(* CODESYS project GW42_TVD2300068.project

Project tree, tasks and I/O mapping:
  Device : eSMART (Linux), Exor International, version 3.5.12.0
    application Application
      libraries: Standard, * (System); SysCom, * (System)
      task MainTask (cyclic, interval 20 ms, priority 1) calls PLC_PRG
      program PLC_PRG [ST]: ioList1, digitalProcessing, analogProcessing, commReset, alarmOut, alarmInh, smart_ship
      Symbols
      function block fb_alarmEvent [ST]
      global variables GVL1
      function block fb_tankMonitor [ST]
      function block fb_scaling20R [ST]
      function block fb_linScaleR [ST]
      function block sh_2 [ST]
      function block fb_fluctDet [ST]
      function block fb_nonLinScale20 [ST]
      function block fb_h2s [ST]
      function block fb_buzzer [ST]
      function block fb_comAlarm [ST]
      function block fb_tankMonitor_magLt [ST]
      function block commCheck [ST]
    Modbus_COM : Modbus COM, 3S - Smart Software Solutions GmbH, version 3.5.15.0
      Modbus_Master_COM_Port : Modbus Master, COM Port, 3S - Smart Software Solutions GmbH, version 3.5.15.0
          settings: Transmission = 'RTU'; ResponseTimeout = 1000; TimeBetweenFrames = 5; Auto-restart communication = TRUE
        Modbus_Slave_im1 : Modbus Slave, COM Port, 3S - Smart Software Solutions GmbH, version 3.5.15.0
            settings: SlaveAddress = 11; Channel 0.Function Code = 3; Channel 0.Read Offset = 16#0007; Channel 0.Read Length = 1; Channel 0.Write Offset = 0; Channel 0.Write Length = 0; Channel 0.Cycle Time = 100; Channel 1.Function Code = 3; Channel 1.Read Offset = 16#0064; Channel 1.Read Length = 1; Channel 1.Write Offset = 0; Channel 1.Write Length = 0; Channel 1.Cycle Time = 100
            input  im1model : WORD  // Channel 0.Channel 0
            input  w_im1IOstatus : WORD  // Channel 1.Channel 1
            unmapped channels: Channel 0, Channel 1
        Modbus_Slave_im2 : Modbus Slave, COM Port, 3S - Smart Software Solutions GmbH, version 3.5.15.0
            settings: SlaveAddress = 12; Channel 0.Function Code = 3; Channel 0.Read Offset = 16#0007; Channel 0.Read Length = 1; Channel 0.Write Offset = 0; Channel 0.Write Length = 0; Channel 0.Cycle Time = 100; Channel 1.Function Code = 3; Channel 1.Read Offset = 16#0064; Channel 1.Read Length = 1; Channel 1.Write Offset = 0; Channel 1.Write Length = 0; Channel 1.Cycle Time = 100
            input  im2model : WORD  // Channel 0.Channel 0
            input  w_im2IOstatus : WORD  // Channel 1.Channel 1
            unmapped channels: Channel 0, Channel 1
        Modbus_Slave_im3 : Modbus Slave, COM Port, 3S - Smart Software Solutions GmbH, version 3.5.15.0
            settings: SlaveAddress = 13; Channel 0.Function Code = 3; Channel 0.Read Offset = 16#0007; Channel 0.Read Length = 1; Channel 0.Write Offset = 0; Channel 0.Write Length = 0; Channel 0.Cycle Time = 100; Channel 1.Function Code = 3; Channel 1.Read Offset = 16#0064; Channel 1.Read Length = 1; Channel 1.Write Offset = 0; Channel 1.Write Length = 0; Channel 1.Cycle Time = 100
            input  im3model : WORD  // Channel 0.Channel 0
            input  w_im3IOstatus : WORD  // Channel 1.Channel 1
            unmapped channels: Channel 0, Channel 1
        Modbus_Slave_im4 : Modbus Slave, COM Port, 3S - Smart Software Solutions GmbH, version 3.5.15.0
            settings: SlaveAddress = 14; Channel 0.Function Code = 3; Channel 0.Read Offset = 16#0007; Channel 0.Read Length = 1; Channel 0.Write Offset = 0; Channel 0.Write Length = 0; Channel 0.Cycle Time = 100; Channel 1.Function Code = 3; Channel 1.Read Offset = 16#0064; Channel 1.Read Length = 1; Channel 1.Write Offset = 0; Channel 1.Write Length = 0; Channel 1.Cycle Time = 100
            input  im4model : WORD  // Channel 0.Channel 0
            input  w_im4IOstatus : WORD  // Channel 1.Channel 1
            unmapped channels: Channel 0, Channel 1
        Modbus_Slave_im5 : Modbus Slave, COM Port, 3S - Smart Software Solutions GmbH, version 3.5.15.0
            settings: SlaveAddress = 15; Channel 0.Function Code = 3; Channel 0.Read Offset = 16#0007; Channel 0.Read Length = 1; Channel 0.Write Offset = 0; Channel 0.Write Length = 0; Channel 0.Cycle Time = 100; Channel 1.Function Code = 3; Channel 1.Read Offset = 16#0064; Channel 1.Read Length = 1; Channel 1.Write Offset = 0; Channel 1.Write Length = 0; Channel 1.Cycle Time = 100
            input  im5model : WORD  // Channel 0.Channel 0
            input  w_im5IOstatus : WORD  // Channel 1.Channel 1
            unmapped channels: Channel 0, Channel 1
        Modbus_Slave_im6 : Modbus Slave, COM Port, 3S - Smart Software Solutions GmbH, version 3.5.15.0
            settings: SlaveAddress = 16; Channel 0.Function Code = 3; Channel 0.Read Offset = 16#0007; Channel 0.Read Length = 1; Channel 0.Write Offset = 0; Channel 0.Write Length = 0; Channel 0.Cycle Time = 100; Channel 1.Function Code = 3; Channel 1.Read Offset = 16#0064; Channel 1.Read Length = 1; Channel 1.Write Offset = 0; Channel 1.Write Length = 0; Channel 1.Cycle Time = 100
            input  im6model : WORD  // Channel 0.Channel 0
            input  w_im6IOstatus : WORD  // Channel 1.Channel 1
            unmapped channels: Channel 0, Channel 1
        Modbus_Slave_im7 : Modbus Slave, COM Port, 3S - Smart Software Solutions GmbH, version 3.5.15.0
            settings: SlaveAddress = 17; Channel 0.Function Code = 3; Channel 0.Read Offset = 16#0007; Channel 0.Read Length = 1; Channel 0.Write Offset = 0; Channel 0.Write Length = 0; Channel 0.Cycle Time = 100; Channel 1.Function Code = 3; Channel 1.Read Offset = 16#0064; Channel 1.Read Length = 1; Channel 1.Write Offset = 0; Channel 1.Write Length = 0; Channel 1.Cycle Time = 100
            input  im7model : WORD  // Channel 0.Channel 0
            input  w_im7IOstatus : WORD  // Channel 1.Channel 1
            unmapped channels: Channel 0, Channel 1
        Modbus_Slave_om1 : Modbus Slave, COM Port, 3S - Smart Software Solutions GmbH, version 3.5.15.0
            settings: SlaveAddress = 21; ResponseTimeout = 1000; UseExtendedFunctionCodes = TRUE; Channel 0.Function Code = 3; Channel 0.Read Offset = 16#0007; Channel 0.Read Length = 1; Channel 0.Write Offset = 0; Channel 0.Write Length = 0; Channel 0.Cycle Time = 100; Channel 1.Function Code = 6; Channel 1.Read Offset = 0; Channel 1.Read Length = 0; Channel 1.Write Offset = 16#0064; Channel 1.Write Length = 1; Channel 1.Cycle Time = 100
            input  om1model : WORD  // Channel 0.Channel 0
            output w_om1IOStatus : WORD  // Channel 1.Channel 1
            unmapped channels: Channel 0, Channel 1
        Modbus_Slave_aim1 : Modbus Slave, COM Port, 3S - Smart Software Solutions GmbH, version 3.5.15.0
            settings: SlaveAddress = 22; ResponseTimeout = 1000; UseExtendedFunctionCodes = TRUE; Channel 0.Function Code = 3; Channel 0.Read Offset = 16#0007; Channel 0.Read Length = 1; Channel 0.Write Offset = 0; Channel 0.Write Length = 0; Channel 0.Cycle Time = 100; Channel 1.Function Code = 3; Channel 1.Read Offset = 16#0064; Channel 1.Read Length = 16; Channel 1.Write Offset = 0; Channel 1.Write Length = 0; Channel 1.Cycle Time = 100
            input  aim1model : WORD  // Channel 0.Channel 0
            input  w_aim1ch1 : WORD  // Channel 1.Channel 1
            input  w_aim1ch2 : WORD  // Channel 1.Channel 1
            input  w_aim1ch3 : WORD  // Channel 1.Channel 1
            input  w_aim1ch4 : WORD  // Channel 1.Channel 1
            input  w_aim1ch5 : WORD  // Channel 1.Channel 1
            input  w_aim1ch6 : WORD  // Channel 1.Channel 1
            input  w_aim1ch7 : WORD  // Channel 1.Channel 1
            input  w_aim1ch8 : WORD  // Channel 1.Channel 1
            input  w_aim1ch9 : WORD  // Channel 1.Channel 1
            input  w_aim1ch10 : WORD  // Channel 1.Channel 1
            input  w_aim1ch11 : WORD  // Channel 1.Channel 1
            input  w_aim1ch12 : WORD  // Channel 1.Channel 1
            input  w_aim1ch13 : WORD  // Channel 1.Channel 1
            input  w_aim1ch14 : WORD  // Channel 1.Channel 1
            input  w_aim1ch15 : WORD  // Channel 1.Channel 1
            input  w_aim1ch16 : WORD  // Channel 1.Channel 1
            unmapped channels: Channel 0, Channel 1
        Modbus_Slave_iom1 : Modbus Slave, COM Port, 3S - Smart Software Solutions GmbH, version 3.5.15.0
            settings: SlaveAddress = 20; ResponseTimeout = 1000; UseExtendedFunctionCodes = TRUE; Channel 0.Function Code = 3; Channel 0.Read Offset = 16#0007; Channel 0.Read Length = 1; Channel 0.Write Offset = 0; Channel 0.Write Length = 0; Channel 0.Cycle Time = 100; Channel 1.Function Code = 3; Channel 1.Read Offset = 16#0064; Channel 1.Read Length = 1; Channel 1.Write Offset = 0; Channel 1.Write Length = 0; Channel 1.Cycle Time = 100; Channel 2.Function Code = 6; Channel 2.Read Offset = 0; Channel 2.Read Length = 0; Channel 2.Write Offset = 16#0065; Channel 2.Write Length = 1; Channel 2.Cycle Time = 100
            input  iom1model : WORD  // Channel 0.Channel 0
            input  w_iom1Istatus : WORD  // Channel 1.Channel 1
            output w_iom1OStatus : WORD  // Channel 2.Channel 2
            unmapped channels: Channel 0, Channel 1, Channel 2
        Modbus_Slave_im9 : Modbus Slave, COM Port, 3S - Smart Software Solutions GmbH, version 3.5.15.0
            settings: SlaveAddress = 19; ResponseTimeout = 1000; UseExtendedFunctionCodes = TRUE; Channel 0.Function Code = 3; Channel 0.Read Offset = 16#0007; Channel 0.Read Length = 1; Channel 0.Write Offset = 0; Channel 0.Write Length = 0; Channel 0.Cycle Time = 100; Channel 1.Function Code = 3; Channel 1.Read Offset = 16#0064; Channel 1.Read Length = 1; Channel 1.Write Offset = 0; Channel 1.Write Length = 0; Channel 1.Cycle Time = 100
            input  im9model : WORD  // Channel 0.Channel 0
            input  w_im9IOstatus : WORD  // Channel 1.Channel 1
            unmapped channels: Channel 0, Channel 1
        Modbus_Slave_im8 : Modbus Slave, COM Port, 3S - Smart Software Solutions GmbH, version 3.5.15.0
            settings: SlaveAddress = 18; ResponseTimeout = 1000; UseExtendedFunctionCodes = TRUE; Channel 0.Function Code = 3; Channel 0.Read Offset = 16#0007; Channel 0.Read Length = 1; Channel 0.Write Offset = 0; Channel 0.Write Length = 0; Channel 0.Cycle Time = 100; Channel 1.Function Code = 3; Channel 1.Read Offset = 16#0064; Channel 1.Read Length = 1; Channel 1.Write Offset = 0; Channel 1.Write Length = 0; Channel 1.Cycle Time = 100
            input  im8model : WORD  // Channel 0.Channel 0
            input  w_im8IOstatus : WORD  // Channel 1.Channel 1
            unmapped channels: Channel 0, Channel 1
    Ethernet : Ethernet, 3S - Smart Software Solutions GmbH, version 3.5.15.0
        settings: IPAddress = [192,168,2,141]; SubnetMask = [255,255,255,0]; GatewayAddress = [0,0,0,0]; MACAddress = [16#00,16#30,16#D8,16#0D,16#B1,16#39]; NetworkInterfaceName = 'eth0'; NetworkInterfaceName = "eth0"; SaveCommunicationSettings = FALSE
      ModbusTCP_Slave_Device : ModbusTCP Slave Device, 3S - Smart Software Solutions GmbH, version 3.5.15.0
          settings: Unit-ID = 1
          output JB1_DATA : WORD  // Outputs.Outputs
          output JB2_DATA : WORD  // Outputs.Outputs
          output JB3_DATA : WORD  // Outputs.Outputs
          output JB4_DATA : WORD  // Outputs.Outputs
          output JB5_DATA : WORD  // Outputs.Outputs
          output JB6_DATA : WORD  // Outputs.Outputs
          output WH_DATA : WORD  // Outputs.Outputs
          output MP1_DATA : WORD  // Outputs.Outputs
          output MP2_DATA : WORD  // Outputs.Outputs
          output MP3_DATA : WORD  // Outputs.Outputs
          output AI1_DATA : WORD  // Outputs.Outputs
          output AI2_DATA : WORD  // Outputs.Outputs
          output AI3_DATA : WORD  // Outputs.Outputs
          output AI4_DATA : WORD  // Outputs.Outputs
          output AI5_DATA : WORD  // Outputs.Outputs
          output AI6_DATA : WORD  // Outputs.Outputs
          output AI7_DATA : WORD  // Outputs.Outputs
          output AI8_DATA : WORD  // Outputs.Outputs
          output AI9_DATA : WORD  // Outputs.Outputs
          output AI10_DATA : WORD  // Outputs.Outputs
          output AI11_DATA : WORD  // Outputs.Outputs
          output AI12_DATA : WORD  // Outputs.Outputs
          output AI13_DATA : WORD  // Outputs.Outputs
          output AI14_DATA : WORD  // Outputs.Outputs
          output COM_DATA : WORD  // Outputs.Outputs
          unmapped channels: Inputs, Outputs
*)

// Device/Application/GVL1
{attribute 'qualified_only'}
VAR_GLOBAL
	hxi_ack	:	BOOL;
	hxi_silence	:	BOOL;
	hxi_ackEr	:	BOOL;
	hxi_silenceEr	:	BOOL;
	hxi_ackWh	:	BOOL;
	hxi_ackWhOut	:	BOOL;
	hxi_silenceWh	:	BOOL;
	hxi_ackMess	:	BOOL;
	hxi_ackMessOut	:	BOOL;
	hxi_silenceMess	:	BOOL;
	hxo_alarmInd	:	BOOL;
	hxo_alarmIndwh	:	BOOL;
	hxo_alarmIndMess	:	BOOL;
	hxi_alarmInh	:	ARRAY[0..310]	OF	BOOL;
	hxo_inhibited	:	BOOL;
	hwo_inhibited	:	WORD;
	hxi_enginesd_accept: BOOL;
	hxi_enginesd_overide: BOOL;
	hwi_override :WORD;
	enginesd_cd: TIME;
    hxi_inhbit_doors: BOOL;
	Hbo_HMITest: BOOL;
	Hbi_HMI1Resp: BOOL;
	Hbi_HMI2Resp: BOOL;
	Hbi_HMI3Resp: BOOL;
	(**)
	pwi_digitalInputs		: ARRAY[0..12]	OF	WORD;
	pwo_digitalOutputs		: ARRAY[0..4] OF WORD;
	hwi_digAlarmSet		: ARRAY[0..12]	OF	WORD;
	hwi_digAlarmDelay0	: ARRAY[0..15] OF WORD;
	hwi_digAlarmDelay1	: ARRAY[0..15] OF WORD;
	hwi_digAlarmDelay2	: ARRAY[0..15] OF WORD;
	hwi_digAlarmDelay3	: ARRAY[0..15] OF WORD;
	hwi_digAlarmDelay4	: ARRAY[0..15] OF WORD;
	hwi_digAlarmDelay5	: ARRAY[0..15] OF WORD;
	hwi_digAlarmDelay6	: ARRAY[0..15] OF WORD;
	hwi_digAlarmDelay7	: ARRAY[0..15] OF WORD;
	hwi_digAlarmDelay8	: ARRAY[0..15] OF WORD;
	hwi_digAlarmDelay9	: ARRAY[0..15] OF WORD;
	hwi_digAlarmDelay10	: ARRAY[0..15] OF WORD;
	hwi_digAlarmDelay11	: ARRAY[0..15] OF WORD;
	hwi_digAlarmDelay12	: ARRAY[0..15] OF WORD;
	hwi_digAlarmInh		: ARRAY[0..12]	OF	WORD;
	hwi_digAlarmOrEvent		: ARRAY[0..12]	OF	WORD;
	hwo_digitalAlarms		: ARRAY[0..12]	OF	WORD;
	hwo_digitalEvents		: ARRAY[0..12]	OF	WORD;
	hwo_digitalAlarmsp		: ARRAY[0..12]	OF	WORD;
	(**)
	pwi_analogInput	: ARRAY[0..15]	OF	WORD;
	hro_ch0OutVal	: ARRAY[0..5] OF REAL;
	hro_ch1OutVal	: ARRAY[0..5] OF REAL;
	hro_ch2OutVal	: ARRAY[0..5] OF REAL;
	hro_ch3OutVal	: ARRAY[0..5] OF REAL;
	hro_ch4OutVal	: ARRAY[0..5] OF REAL;
	hro_ch5OutVal	: ARRAY[0..5] OF REAL;
	hro_ch6OutVal	: ARRAY[0..5] OF REAL;
	hro_ch7OutVal	: ARRAY[0..5] OF REAL;
	hro_ch8OutVal	: ARRAY[0..5] OF REAL;
	hro_ch9OutVal	: ARRAY[0..5] OF REAL;
	hro_ch10OutVal	: ARRAY[0..5] OF REAL;
	hro_ch11OutVal	: ARRAY[0..5] OF REAL;
	hro_ch12OutVal	: ARRAY[0..5] OF REAL;
	hro_ch13OutVal	: ARRAY[0..5] OF REAL;
	hro_ch14OutVal	: ARRAY[0..5] OF REAL;
	hro_ch15OutVal	: ARRAY[0..5] OF REAL;
	(*Analolg channel LIMIT steady alarms AND channel errors TO HMI*)
(*Hwo_AnalogAlm_Ch1G1.0 : Level 1, Hwo_AnalogAlm_Ch1G1.1 : Level 2, Hwo_AnalogAlm_Ch1G1.2 : Level 3,Hwo_AnalogAlm_Ch1G1.3 : Cable break,Hwo_AnalogAlm_Ch1G1.4 : Over range*)

	hwo_analogAlm	: ARRAY[0..15]	OF	WORD;
	(*Analolg channel limit pulse alarms and channel errors to HMI*)
(*Hwo_AnalogAlm_Ch1G1.0 : Level 1, Hwo_AnalogAlm_Ch1G1.1 : Level 2, Hwo_AnalogAlm_Ch1G1.2 : Level 3,Hwo_AnalogAlm_Ch1G1.3 : Cable break,Hwo_AnalogAlm_Ch1G1.4 : Over range*)

	hwo_analogAlmP	: ARRAY[0..15]	OF	WORD;
(*Alarm message*)
	hwo_almMsg	: ARRAY[0..15] OF WORD; (*Tanks*)
	(*Analog alarm inhibition*)
(*0:inhL1, 1:inhL2, 2:inhL3, 3:inhCable break, 4:inhOver range, 5:buz en L1, 6:buz en L2, 7:buz en L3, 8:buz en err1, 9:buz en err2, 10:inhL4, 11:buz en L4, 12: Auto filter enable
							13:Fill input sensor min value and range when tank empty, 14: Fill input sensor max value and range when tank full*)
	hwi_chPara	: ARRAY[0..15]	OF	WORD;
(* Prameters of analog limit and eror alarms to HMI *)
(*0:L1Lt, 1:L2Lt, 2:L3Lt, 3:L1delay, 4:L2delay, 5:L3delay,6:Errdelay,
											7:ErrFactor, 8:SensorValMin,9:SensorValMax, 10:SensorRangeMin, 11:SensorRangeMax, 12:filterVal, 
											13:L4Lt, 14:L4delay, 15:heightMin, 16:heightMax, 17:density, 18:unusable , 19:height offset in mm, 
											Auto filter-->20: rate of change, 21: sampling time, 22:sample hold time, 23:filter time constant*)
	hri_chSP_Ch0	: ARRAY[0..23] OF REAL;
	hri_chSP_Ch1	: ARRAY[0..23] OF REAL;
	hri_chSP_Ch2	: ARRAY[0..23] OF REAL;
	hri_chSP_Ch3	: ARRAY[0..23] OF REAL;
	hri_chSP_Ch4	: ARRAY[0..23] OF REAL;
	hri_chSP_Ch5	: ARRAY[0..23] OF REAL;
	hri_chSP_Ch6	: ARRAY[0..23] OF REAL;
	hri_chSP_Ch7	: ARRAY[0..23] OF REAL;
	hri_chSP_Ch8	: ARRAY[0..23] OF REAL;
	hri_chSP_Ch9	: ARRAY[0..23] OF REAL;
	hri_chSP_Ch10	: ARRAY[0..23] OF REAL;
	hri_chSP_Ch11	: ARRAY[0..23] OF REAL;
	hri_chSP_Ch12	: ARRAY[0..23] OF REAL;
	hri_chSP_Ch13	: ARRAY[0..23] OF REAL;
	hri_chSP_Ch14	: ARRAY[0..23] OF REAL;
	hri_chSP_Ch15	: ARRAY[0..23] OF REAL;
(*Tank level sampling in*)
	hwi_ch0X	: ARRAY[0..20] OF WORD;
	hwi_ch1X	: ARRAY[0..20] OF WORD;
	hwi_ch2X	: ARRAY[0..20] OF WORD;
	hwi_ch3X	: ARRAY[0..20] OF WORD;
	hwi_ch4X	: ARRAY[0..20] OF WORD;	
	hwi_ch5X	: ARRAY[0..20] OF WORD;	
	hwi_ch6X	: ARRAY[0..20] OF WORD;	
	hwi_ch7X	: ARRAY[0..20] OF WORD;	
	hwi_ch8X	: ARRAY[0..20] OF WORD;	
	hwi_ch9X	: ARRAY[0..20] OF WORD;	
	hwi_ch10X	: ARRAY[0..20] OF WORD;	
	hwi_ch11X	: ARRAY[0..20] OF WORD;	
	hwi_ch12X	: ARRAY[0..20] OF WORD;	
	hwi_ch13X	: ARRAY[0..20] OF WORD;	
	hwi_ch14X	: ARRAY[0..20] OF WORD;	
	hwi_ch15X	: ARRAY[0..20] OF WORD;	
(*Tank level sampling out*)
	hwi_ch0Y	: ARRAY[0..20] OF WORD;
	hwi_ch1Y	: ARRAY[0..20] OF WORD;
	hwi_ch2Y	: ARRAY[0..20] OF WORD;
	hwi_ch3Y	: ARRAY[0..20] OF WORD;
	hwi_ch4Y	: ARRAY[0..20] OF WORD;
	hwi_ch5Y	: ARRAY[0..20] OF WORD;
	hwi_ch6Y	: ARRAY[0..20] OF WORD;
	hwi_ch7Y	: ARRAY[0..20] OF WORD;
	hwi_ch8Y	: ARRAY[0..20] OF WORD;
	hwi_ch9Y	: ARRAY[0..20] OF WORD;
	hwi_ch10Y	: ARRAY[0..20] OF WORD;
	hwi_ch11Y	: ARRAY[0..20] OF WORD;	
	hwi_ch12Y	: ARRAY[0..20] OF WORD;	
	hwi_ch13Y	: ARRAY[0..20] OF WORD;	
	hwi_ch14Y	: ARRAY[0..20] OF WORD;	
	hwi_ch15Y	: ARRAY[0..20] OF WORD;			

END_VAR

// Device/Application/PLC_PRG
PROGRAM PLC_PRG
VAR
	w_modelNo1 : WORD;
	w_modelNo2 : WORD;
	w_modelNo3 : WORD;
	(**)
	aeGroup0: fb_alarmEvent;
	aeGroup1: fb_alarmEvent;
	aeGroup2: fb_alarmEvent;
	aeGroup3: fb_alarmEvent;
	aeGroup4: fb_alarmEvent;
	aeGroup5: fb_alarmEvent;
	aeGroup6: fb_alarmEvent;
	aeGroup7: fb_alarmEvent;
	aeGroup8: fb_alarmEvent;
	aeGroup9: fb_alarmEvent;
	aeGroup10: fb_alarmEvent;
	aeGroup11: fb_alarmEvent;
	aeGroup12: fb_alarmEvent;
	
	w_digAlarmInh		: ARRAY[0..12]	OF	WORD;
	w_anaAlarmInh		: ARRAY[0..15]	OF	WORD;
	lwi_interlocks		: ARRAY[0..12]	OF	WORD;
	lx_refresh: BOOL;
	lx_ack: BOOL;
	lwo_dialmBuzzer: WORD;
	lwo_dialmInd: WORD;
	(**)
	tmGroup0: fb_tankMonitor;	
	tmGroup1: fb_tankMonitor;
	tmGroup2: fb_tankMonitor;
	tmGroup3: fb_tankMonitor;
	tmGroup4: fb_tankMonitor;
	tmGroup5: fb_tankMonitor;
	tmGroup6: fb_tankMonitor;
	tmGroup7: fb_tankMonitor;
	tmGroup8: fb_tankMonitor;
	tmGroup9: fb_tankMonitor;
	tmGroup10: fb_tankMonitor;
	tmGroup11: fb_tankMonitor;	
	tmGroup12: fb_tankMonitor;
	tmGroup13: fb_tankMonitor;
	tmGroup14: fb_tankMonitor;
	tmGroup15: fb_tankMonitor;	
	lwo_aialmBuzzer: WORD;
	lwo_aialmInd: WORD;
	
	
(*commReset*)	
	x_im1Error : BOOL;
	im1Errorcode : MB_ErrorCodes;
	x_im1Ack: BOOL;

	x_masterReset: BOOL;
	x_im1Reset: BOOL;
	x_im2Reset: BOOL;
	x_im3Reset: BOOL;
	x_im4Reset: BOOL;
	x_im5Reset: BOOL;
	x_im6Reset: BOOL;
	x_im7Reset: BOOL;
	x_im8Reset: BOOL;
	x_om1Reset: BOOL;
	x_aim1Reset: BOOL;	
	
	ton_blink1: TON;
	ton_blink2: TON;
	ton_blink3: TON;
	ton_blink4: TON;
	ton_blink5: TON;
	ton_blink6: TON;
	ton_blink7: TON;
	ton_blink8: TON;
	ton_blink9: TON;
	ton_blink11: TON;
	ton_blink12: TON;
	ton_blink13: TON;
	ton_blink14: TON;
	ton_blink15: TON;
	ton_blink16: TON;
	ton_blink17: TON;
	ton_blink18: TON;
	ton_blink19: TON;
	ton_blink20: TON;
	ton_blink21: TON;	
	ton_blink22: TON;
	
	tp_blink1: TP;
	tp_blink2: TP;
	tp_blink3: TP;
	tp_blink4: TP;
	tp_blink5: TP;
	tp_blink6: TP;
	tp_blink7: TP;
	tp_blink8: TP;
	tp_blink9: TP;
	tp_blink10: TP;
	tp_blink11: TP;
	tp_blink12: TP;
	tp_blink13: TP;
	tp_blink14: TP;
	tp_blink15: TP;
	tp_blink16: TP;
	tp_blink17: TP;
	tp_blink18: TP;
	tp_blink19: TP;
	tp_blink20: TP;
	tp_blink21: TP;
	tp_blink22: TP;
	

	x_mbReset: BOOL;
(*Alarm out*)
	buzzerSet1: fb_buzzer;
	buzzerSet2: fb_buzzer;
	buzzerSet3: fb_buzzer;
	buzzerSet4: fb_buzzer;
	buzzerSet5: fb_buzzer;
    buzzerSet6: fb_buzzer;			
	comAlarm: fb_comAlarm;
	comAlarm1: fb_comAlarm;
	comAlarm2: fb_comAlarm;	
commCheck1: commCheck;
	ee: fb_tankMonitor;
	ton_enginesd: TON;
	
	
	
	overide_out: BOOL;
	poweron_ton: TON;
	wi_interlocks: INT;
END_VAR

w_modelNo1 := im1model;

ioList1();
digitalProcessing();
analogProcessing();
alarmOut();
commReset();
alarmInh();
smart_ship();

ACTION ioList1:
//Digital input module JB1 - S3306: 16CH							
GVL1.Pwi_DigitalInputs[0].0	 := NOT w_im1IOStatus.0	AND NOT GVL1.hwo_digitalAlarms[12].0	;	(*	DI:01	GEN.ROOM PORT BILGE ALARM	*)
GVL1.Pwi_DigitalInputs[0].1	 := NOT w_im1IOStatus.1	AND NOT GVL1.hwo_digitalAlarms[12].0	;	(*	DI:02	PORT GEN EXHAUST TEMP HIGH	*)
GVL1.Pwi_DigitalInputs[0].2	 := NOT w_im1IOStatus.2	AND NOT GVL1.hwo_digitalAlarms[12].0	;	(*	DI:03	PORT GENERATOR COMMON ALARM	*)
GVL1.Pwi_DigitalInputs[0].3	 := NOT w_im1IOStatus.3	AND NOT GVL1.hwo_digitalAlarms[12].0	;	(*	DI:04	PORT GENERATOR RUNNING INDICATION	*)
GVL1.Pwi_DigitalInputs[0].4	 := NOT w_im1IOStatus.4	AND NOT GVL1.hwo_digitalAlarms[12].0	;	(*	DI:05	A.FOULING ALARM: DG(P) & EMG FIRE.P S/C 	*)
GVL1.Pwi_DigitalInputs[0].5	 := NOT w_im1IOStatus.5	AND NOT GVL1.hwo_digitalAlarms[12].0	;	(*	DI:06	STEERING CP: PHASE FAIL MOTOR 1	*)
GVL1.Pwi_DigitalInputs[0].6	 := NOT w_im1IOStatus.6	AND NOT GVL1.hwo_digitalAlarms[12].0	;	(*	DI:07	STEERING CP: POWER FAIL MOTOR 1	*)
GVL1.Pwi_DigitalInputs[0].7	 := NOT w_im1IOStatus.7	AND NOT GVL1.hwo_digitalAlarms[12].0	;	(*	DI:08	STEERING CP: CONTROL FAIL MOTOR 1	*)
GVL1.Pwi_DigitalInputs[0].8	 := NOT w_im1IOStatus.8	AND NOT GVL1.hwo_digitalAlarms[12].0	;	(*	DI:09	STEERING CP: OVERLOAD MOTOR 1	*)
GVL1.Pwi_DigitalInputs[0].9	 := NOT w_im1IOStatus.9	AND NOT GVL1.hwo_digitalAlarms[12].0	;	(*	DI:10	STEERING CP: PHASE FAIL MOTOR 2	*)
GVL1.Pwi_DigitalInputs[0].10	 := NOT w_im1IOStatus.10	AND NOT GVL1.hwo_digitalAlarms[12].0	;	(*	DI:11	STEERING CP: POWER FAIL MOTOR 2	*)
GVL1.Pwi_DigitalInputs[0].11	 := NOT w_im1IOStatus.11	AND NOT GVL1.hwo_digitalAlarms[12].0	;	(*	DI:12	STEERING CP: CONTROL FAIL MOTOR 2	*)
GVL1.Pwi_DigitalInputs[0].12	 := NOT w_im1IOStatus.12	AND NOT GVL1.hwo_digitalAlarms[12].0	;	(*	DI:13	STEERING CP: OVERLOAD MOTOR 2	*)
GVL1.Pwi_DigitalInputs[0].13	 := NOT w_im1IOStatus.13	AND NOT GVL1.hwo_digitalAlarms[12].0	;	(*	DI:14	STEERING CP: LOW OIL LEVEL ALARM	*)
GVL1.Pwi_DigitalInputs[0].14	 := NOT w_im1IOStatus.14	AND NOT GVL1.hwo_digitalAlarms[12].0	;	(*	DI:15	STEERING CP: HIGH OIL TEMP ALARM	*)
GVL1.Pwi_DigitalInputs[0].15	 := NOT w_im1IOStatus.15	AND NOT GVL1.hwo_digitalAlarms[12].0	;	(*	DI:16	STEERING CP: LOW OIL PRESSURE ALARM	*)
//Digital input module JB2 - S3306: 16CH							
GVL1.Pwi_DigitalInputs[1].0	 := NOT w_im2IOStatus.0	AND NOT GVL1.hwo_digitalAlarms[12].1	;	(*	DI:17	GEN.ROOM STBD BILGE ALARM	*)
GVL1.Pwi_DigitalInputs[1].1	 := NOT w_im2IOStatus.1	AND NOT GVL1.hwo_digitalAlarms[12].1	;	(*	DI:18	ENGINE ROOM AFT WT DOOR	*)
GVL1.Pwi_DigitalInputs[1].2	 := NOT w_im2IOStatus.2	AND NOT GVL1.hwo_digitalAlarms[12].1	;	(*	DI:19	CENTER ME EXHAUST TEMP HIGH	*)
GVL1.Pwi_DigitalInputs[1].3	 := NOT w_im2IOStatus.3	AND NOT GVL1.hwo_digitalAlarms[12].1	;	(*	DI:20	STBD GEN EXHAUST TEMP HIGH	*)
GVL1.Pwi_DigitalInputs[1].4	 := NOT w_im2IOStatus.4	AND NOT GVL1.hwo_digitalAlarms[12].1	;	(*	DI:21	STBD GENERATOR COMMON ALARM	*)
GVL1.Pwi_DigitalInputs[1].5	 := NOT w_im2IOStatus.5	AND NOT GVL1.hwo_digitalAlarms[12].1	;	(*	DI:22	STBD GENERATOR RUNNING INDICATION	*)
GVL1.Pwi_DigitalInputs[1].6	 := NOT w_im2IOStatus.6	AND NOT GVL1.hwo_digitalAlarms[12].1	;	(*	DI:23	STBD ME EXHAUST TEMP HIGH	*)
GVL1.Pwi_DigitalInputs[1].7	 := NOT w_im2IOStatus.7	AND NOT GVL1.hwo_digitalAlarms[12].1	;	(*	DI:24	BOW THRUSTER COMMON ALARM	*)
GVL1.Pwi_DigitalInputs[1].8	 := NOT w_im2IOStatus.8	AND NOT GVL1.hwo_digitalAlarms[12].1	;	(*	DI:25	BOW THRUSTER LOW OIL LEVEL ALARM	*)
GVL1.Pwi_DigitalInputs[1].9	 := NOT w_im2IOStatus.9	AND NOT GVL1.hwo_digitalAlarms[12].1	;	(*	DI:26	BOW THRUSTER HIGH OIL TEMP ALARM	*)
GVL1.Pwi_DigitalInputs[1].10	:= NOT w_im2IOStatus.10	AND NOT GVL1.hwo_digitalAlarms[12].1	;	(*	DI:27	OWS POWER SUPPLY FAILURE	*)
GVL1.Pwi_DigitalInputs[1].11	:= NOT w_im2IOStatus.11	AND NOT GVL1.hwo_digitalAlarms[12].1	;	(*	DI:28	OWS 15 PPM ALARM	*)
GVL1.Pwi_DigitalInputs[1].12	:= NOT w_im2IOStatus.12	AND NOT GVL1.hwo_digitalAlarms[12].1	;	(*	DI:29	DCDB-2 BATTERY BREAKER TRIP ALARM	*)
GVL1.Pwi_DigitalInputs[1].13	:= NOT w_im2IOStatus.13	AND NOT GVL1.hwo_digitalAlarms[12].1	;	(*	DI:30	DCDB-2 EARTH FAULT ALARM	*)
GVL1.Pwi_DigitalInputs[1].14	:= NOT w_im2IOStatus.14	AND NOT GVL1.hwo_digitalAlarms[12].1	;	(*	DI:31	DCDB-2 BATTERY CHARGER FAIL ALARM	*)
GVL1.Pwi_DigitalInputs[1].15	:= NOT w_im2IOStatus.15	AND NOT GVL1.hwo_digitalAlarms[12].1	;	(*	DI:32	DCDB-2 BATTERY DISCHARGE ALARM	*)
//Digital input module JB3 - S3306: 16CH							
GVL1.Pwi_DigitalInputs[2].0	:= NOT w_im3IOStatus.0	AND NOT GVL1.hwo_digitalAlarms[12].2	;	(*	DI:33	PORT STERN TUBE FLOW ALARM	*)
GVL1.Pwi_DigitalInputs[2].1	:= NOT w_im3IOStatus.1	AND NOT GVL1.hwo_digitalAlarms[12].2	;	(*	DI:34	STBD STERN TUBE FLOW ALARM	*)
GVL1.Pwi_DigitalInputs[2].2	:= NOT w_im3IOStatus.2	AND NOT GVL1.hwo_digitalAlarms[12].2	;	(*	DI:35	CENTER STERN TUBE FLOW ALARM	*)
GVL1.Pwi_DigitalInputs[2].3	:= NOT w_im3IOStatus.3	AND NOT GVL1.hwo_digitalAlarms[12].2	;	(*	DI:36	PORT ME EXHAUST TEMP HIGH	*)
GVL1.Pwi_DigitalInputs[2].4	:= NOT w_im3IOStatus.4	AND NOT GVL1.hwo_digitalAlarms[12].2	;	(*	DI:37	A.FOULING ALARM: AUX SW.P & EMG FIRE.P S/C	*)
GVL1.Pwi_DigitalInputs[2].5	:= NOT w_im3IOStatus.5	AND NOT GVL1.hwo_digitalAlarms[12].2	;	(*	DI:38	A.FOULING ALARM: DG(S) S/C	*)
GVL1.Pwi_DigitalInputs[2].6	:= NOT w_im3IOStatus.6	AND NOT GVL1.hwo_digitalAlarms[12].2	;	(*	DI:39	PORT ME/GEN STARTING BATTERY LOW ALARM	*)
GVL1.Pwi_DigitalInputs[2].7	:= NOT w_im3IOStatus.7	AND NOT GVL1.hwo_digitalAlarms[12].2	;	(*	DI:40	STBD ME/GEN STARTING BATTERY LOW ALARM	*)
GVL1.Pwi_DigitalInputs[2].8	:= NOT w_im3IOStatus.8	AND NOT GVL1.hwo_digitalAlarms[12].2	;	(*	DI:41	CENTER ME STARTING BATTERY LOW ALARM	*)
GVL1.Pwi_DigitalInputs[2].9	:= NOT w_im3IOStatus.9	AND NOT GVL1.hwo_digitalAlarms[12].2	;	(*	DI:42	AUX COOLING PUMP-2 RUNNING	*)
GVL1.Pwi_DigitalInputs[2].10	:= NOT w_im3IOStatus.10	AND NOT GVL1.hwo_digitalAlarms[12].2	;	(*	DI:43	AUX COOLING PUMP-2 TRIP	*)
GVL1.Pwi_DigitalInputs[2].11	:= NOT w_im3IOStatus.11	AND NOT GVL1.hwo_digitalAlarms[12].2	;	(*	DI:44	ENG.ROOM AFT BILGE ALARM	*)
GVL1.Pwi_DigitalInputs[2].12	:= NOT w_im3IOStatus.12	AND NOT GVL1.hwo_digitalAlarms[12].2	;	(*	DI:45	ENG.ROOM AFT FLOOD ALARM	*)
GVL1.Pwi_DigitalInputs[2].13	:= NOT w_im3IOStatus.13	AND NOT GVL1.hwo_digitalAlarms[12].2	;	(*	DI:46	SPARE	*)
GVL1.Pwi_DigitalInputs[2].14	:= NOT w_im3IOStatus.14	AND NOT GVL1.hwo_digitalAlarms[12].2	;	(*	DI:47	SPARE	*)
GVL1.Pwi_DigitalInputs[2].15	:= NOT w_im3IOStatus.15	AND NOT GVL1.hwo_digitalAlarms[12].2	;	(*	DI:48	SPARE	*)
//Digital input module JB4 - S3306: 16CH							
GVL1.Pwi_DigitalInputs[3].0	:= NOT w_im4IOStatus.0	AND NOT GVL1.hwo_digitalAlarms[12].3	;	(*	DI:49	ENG.ROOM FWD BILGE ALARM	*)
GVL1.Pwi_DigitalInputs[3].1	:= NOT w_im4IOStatus.1	AND NOT GVL1.hwo_digitalAlarms[12].3	;	(*	DI:50	ENG.ROOM FWD FLOOD ALARM	*)
GVL1.Pwi_DigitalInputs[3].2	:= NOT w_im4IOStatus.2	AND NOT GVL1.hwo_digitalAlarms[12].3	;	(*	DI:51	ENGINE ROOM FWD WT DOOR	*)
GVL1.Pwi_DigitalInputs[3].3	:= NOT w_im4IOStatus.3	AND NOT GVL1.hwo_digitalAlarms[12].3	;	(*	DI:52	PROPULSION SYSTEM POWER SUPPLY FAIL	*)
GVL1.Pwi_DigitalInputs[3].4	:= NOT w_im4IOStatus.4	AND NOT GVL1.hwo_digitalAlarms[12].3	;	(*	DI:53	PORT ME PROP.MODULE COMMON ALARM	*)
GVL1.Pwi_DigitalInputs[3].5	:= NOT w_im4IOStatus.5	AND NOT GVL1.hwo_digitalAlarms[12].3	;	(*	DI:54	STBD ME PROP.MODULE COMMON ALARM	*)
GVL1.Pwi_DigitalInputs[3].6	:= NOT w_im4IOStatus.6	AND NOT GVL1.hwo_digitalAlarms[12].3	;	(*	DI:55	CENTER ME PROP.MODULE COMMON ALARM	*)
GVL1.Pwi_DigitalInputs[3].7	:= NOT w_im4IOStatus.7	AND NOT GVL1.hwo_digitalAlarms[12].3	;	(*	DI:56	A.FOULING ALARM: PORT ME & STBD ME S/C	*)
GVL1.Pwi_DigitalInputs[3].8	:= NOT w_im4IOStatus.8	AND NOT GVL1.hwo_digitalAlarms[12].3	;	(*	DI:57	A.FOULING ALARM: CENETR ME S/C	*)
GVL1.Pwi_DigitalInputs[3].9	:= NOT w_im4IOStatus.9	AND NOT GVL1.hwo_digitalAlarms[12].3	;	(*	DI:58	A.FOULING ALARM: SW DOMESTIC & A/C.P SC	*)
GVL1.Pwi_DigitalInputs[3].10	:= NOT w_im4IOStatus.10	AND NOT GVL1.hwo_digitalAlarms[12].3	;	(*	DI:59	ENG.ROOM CO2 RELEASE EAVC ALARM	*)
GVL1.Pwi_DigitalInputs[3].11	:= NOT w_im4IOStatus.11	AND NOT GVL1.hwo_digitalAlarms[12].3	;	(*	DI:60	GEN.ROOM CO2 RELEASE EVAC ALARM	*)
GVL1.Pwi_DigitalInputs[3].12	:= NOT w_im4IOStatus.12	AND NOT GVL1.hwo_digitalAlarms[12].3	;	(*	DI:61	CO2 LEAKAGE ALARM	*)
GVL1.Pwi_DigitalInputs[3].13	:= NOT w_im4IOStatus.13	AND NOT GVL1.hwo_digitalAlarms[12].3	;	(*	DI:62	ENG ROOM CO2 RELEASED ALARM	*)
GVL1.Pwi_DigitalInputs[3].14	:= NOT w_im4IOStatus.14	AND NOT GVL1.hwo_digitalAlarms[12].3	;	(*	DI:63	GEN ROOM CO2 RELEASED ALARM	*)
GVL1.Pwi_DigitalInputs[3].15	:= NOT w_im4IOStatus.15	AND NOT GVL1.hwo_digitalAlarms[12].3	;	(*	DI:64	CO2 SYSTEM POWER FAIL ALARM	*)
//Digital input module JB5 - S3306: 16CH							
GVL1.Pwi_DigitalInputs[4].0	:= NOT w_im5IOStatus.0	AND NOT GVL1.hwo_digitalAlarms[12].4	;	(*	DI:65	PUMP ROOM AFT PORT BILGE ALARM	*)
GVL1.Pwi_DigitalInputs[4].1	:= NOT w_im5IOStatus.1	AND NOT GVL1.hwo_digitalAlarms[12].4	;	(*	DI:66	PUMP ROOM AFT STBD BILGE ALARM	*)
GVL1.Pwi_DigitalInputs[4].2	:= NOT w_im5IOStatus.2	AND NOT GVL1.hwo_digitalAlarms[12].4	;	(*	DI:67	V.SPACE PUMP ROOM FWD (P) BILGE ALARM	*)
GVL1.Pwi_DigitalInputs[4].3	:= NOT w_im5IOStatus.3	AND NOT GVL1.hwo_digitalAlarms[12].4	;	(*	DI:68	V.SPACE PUMP ROOM FWD (S) BILGE ALARM	*)
GVL1.Pwi_DigitalInputs[4].4	:= NOT w_im5IOStatus.4	AND NOT GVL1.hwo_digitalAlarms[12].4	;	(*	DI:69	ACCOM.AREA AFT BILGE ALARM	*)
GVL1.Pwi_DigitalInputs[4].5	:= NOT w_im5IOStatus.5	AND NOT GVL1.hwo_digitalAlarms[12].4	;	(*	DI:70	PUMP ROOM FWD WT DOOR	*)
GVL1.Pwi_DigitalInputs[4].6	:= NOT w_im5IOStatus.6	AND NOT GVL1.hwo_digitalAlarms[12].4	;	(*	DI:71	STP OVERFLOW ALARM	*)
GVL1.Pwi_DigitalInputs[4].7	:= NOT w_im5IOStatus.7	AND NOT GVL1.hwo_digitalAlarms[12].4	;	(*	DI:72	A/C SYSTEM COMMON ALARM	*)
GVL1.Pwi_DigitalInputs[4].8	:= NOT w_im5IOStatus.8	AND NOT GVL1.hwo_digitalAlarms[12].4	;	(*	DI:73	ACCOM.AREA FWD BILGE ALARM	*)
GVL1.Pwi_DigitalInputs[4].9	:= NOT w_im5IOStatus.9	AND NOT GVL1.hwo_digitalAlarms[12].4	;	(*	DI:74	FWD PASSAGE BILGE ALARM	*)
GVL1.Pwi_DigitalInputs[4].10	:= NOT w_im5IOStatus.10	AND NOT GVL1.hwo_digitalAlarms[12].4	;	(*	DI:75	FOREPEAK COMPT BILGE ALARM	*)
GVL1.Pwi_DigitalInputs[4].11	:= NOT w_im5IOStatus.11	AND NOT GVL1.hwo_digitalAlarms[12].4	;	(*	DI:76	ACCOM.AREA WT DOOR	*)
GVL1.Pwi_DigitalInputs[4].12	:= NOT w_im5IOStatus.12	AND NOT GVL1.hwo_digitalAlarms[12].4	;	(*	DI:77	A/C FIRE DAMPER CLOSED ALARM	*)
GVL1.Pwi_DigitalInputs[4].13	:= NOT w_im5IOStatus.13	AND NOT GVL1.hwo_digitalAlarms[12].4	;	(*	DI:78	GALLEY VENT OUT FIRE DAMPER CLOSED ALARM	*)
GVL1.Pwi_DigitalInputs[4].14	:= NOT w_im5IOStatus.14	AND NOT GVL1.hwo_digitalAlarms[12].4	;	(*	DI:79	GALLEY VENT IN FIRE DAMPER CLOSED ALARM	*)
GVL1.Pwi_DigitalInputs[4].15	:= NOT w_im5IOStatus.15	AND NOT GVL1.hwo_digitalAlarms[12].4	;	(*	DI:80	GALLEY HD VENT FIRE DAMPER CLOSED ALARM	*)

//Digital input module JB6 - S3306: 16CH							
GVL1.Pwi_DigitalInputs[5].0	:= NOT w_im6IOStatus.0	AND NOT GVL1.hwo_digitalAlarms[12].5	;	(*	DI:81	DCDB1 SEC-1 BAT.CHARGER FAILURE ALARM	*)
GVL1.Pwi_DigitalInputs[5].1	:= NOT w_im6IOStatus.1	AND NOT GVL1.hwo_digitalAlarms[12].5	;	(*	DI:82	DCDB1 SEC-1 BAT. DISCHARGE ALARM	*)
GVL1.Pwi_DigitalInputs[5].2	:= NOT w_im6IOStatus.2	AND NOT GVL1.hwo_digitalAlarms[12].5	;	(*	DI:83	DCDB1 SEC-1 BAT. LOW VOLT ALARM	*)
GVL1.Pwi_DigitalInputs[5].3	:= NOT w_im6IOStatus.3	AND NOT GVL1.hwo_digitalAlarms[12].5	;	(*	DI:84	DCDB1 SEC-1 BAT. BANK CB TRIP ALARM	*)
GVL1.Pwi_DigitalInputs[5].4	:= NOT w_im6IOStatus.4	AND NOT GVL1.hwo_digitalAlarms[12].5	;	(*	DI:85	DCDB1 SEC-2 BAT.CHARGER FAILURE ALARM	*)
GVL1.Pwi_DigitalInputs[5].5	:= NOT w_im6IOStatus.5	AND NOT GVL1.hwo_digitalAlarms[12].5	;	(*	DI:86	DCDB1 SEC-2 BAT. DISCHARGE ALARM	*)
GVL1.Pwi_DigitalInputs[5].6	:= NOT w_im6IOStatus.6	AND NOT GVL1.hwo_digitalAlarms[12].5	;	(*	DI:87	DCDB1 SEC-2 BAT. LOW VOLT ALARM	*)
GVL1.Pwi_DigitalInputs[5].7	:= NOT w_im6IOStatus.7	AND NOT GVL1.hwo_digitalAlarms[12].5	;	(*	DI:88	DCDB1 SEC-2 BAT. BANK CB TRIP ALARM	*)
GVL1.Pwi_DigitalInputs[5].8	:= NOT w_im6IOStatus.8	AND NOT GVL1.hwo_digitalAlarms[12].5	;	(*	DI:89	SEC-1 AND SEC-2 EARTH FAULT	*)
GVL1.Pwi_DigitalInputs[5].9	:= NOT w_im6IOStatus.9	AND NOT GVL1.hwo_digitalAlarms[12].5	;	(*	DI:90	FREEZER CTRL PANEL COMMON ALARM	*)
GVL1.Pwi_DigitalInputs[5].10	:= NOT w_im6IOStatus.10	AND NOT GVL1.hwo_digitalAlarms[12].5	;	(*	DI:91	CHILLER CTRL PANEL COMMON ALARM	*)
GVL1.Pwi_DigitalInputs[5].11	:= NOT w_im6IOStatus.11	AND NOT GVL1.hwo_digitalAlarms[12].5	;	(*	DI:92	MAN TRAP ALARM: FREEZER ROOM	*)
GVL1.Pwi_DigitalInputs[5].12	:= NOT w_im6IOStatus.12	AND NOT GVL1.hwo_digitalAlarms[12].5	;	(*	DI:93	MAN TRAP ALARM: CHILLER ROOM	*)
GVL1.Pwi_DigitalInputs[5].13	:= NOT w_im6IOStatus.13	AND NOT GVL1.hwo_digitalAlarms[12].5	;	(*	DI:94	PUMP RM COMP. AREA AREA REF. LEAKAGE ALARM 	*)
GVL1.Pwi_DigitalInputs[5].14	:= NOT w_im6IOStatus.14	AND NOT GVL1.hwo_digitalAlarms[12].5	;	(*	DI:95	BELOW DECK. AREA AREA REF. LEAKAGE ALARM 	*)
GVL1.Pwi_DigitalInputs[5].15	:= NOT w_im6IOStatus.15	AND NOT GVL1.hwo_digitalAlarms[12].5	;	(*	DI:96	CO2 ROOM FAN TRIP ALARM	*)
//Digital input module WH - S3306: 16CH							
GVL1.Pwi_DigitalInputs[6].0	:= NOT w_im7IOStatus.0	AND NOT GVL1.hwo_digitalAlarms[12].6	;	(*	DI:97	WH ALARM MUTE P/B	*)
GVL1.Pwi_DigitalInputs[6].1	:= NOT w_im7IOStatus.1	AND NOT GVL1.hwo_digitalAlarms[12].6	;	(*	DI:98	STGR JOYSTICK CONTROL FAIL ALARM	*)
GVL1.Pwi_DigitalInputs[6].2	:= NOT w_im7IOStatus.2	AND NOT GVL1.hwo_digitalAlarms[12].6	;	(*	DI:99	GEN.ALARM MAIN SUPPLY FAILURE	*)
GVL1.Pwi_DigitalInputs[6].3	:= NOT w_im7IOStatus.3	AND NOT GVL1.hwo_digitalAlarms[12].6	;	(*	DI:100	GEN.ALARM ALT.SUPPLY FAILURE	*)
GVL1.Pwi_DigitalInputs[6].4	:= NOT w_im7IOStatus.4	AND NOT GVL1.hwo_digitalAlarms[12].6	;	(*	DI:101	NAV.LIGHT POWER FAILURE	*)
GVL1.Pwi_DigitalInputs[6].5	:= NOT w_im7IOStatus.5	AND NOT GVL1.hwo_digitalAlarms[12].6	;	(*	DI:102	NAV.LIGHT SYSTEM FAULT	*)
GVL1.Pwi_DigitalInputs[6].6	:= NOT w_im7IOStatus.6	AND NOT GVL1.hwo_digitalAlarms[12].6	;	(*	DI:103	FIRE ALARM SYSTEM FAULT	*)
GVL1.Pwi_DigitalInputs[6].7	:= NOT w_im7IOStatus.7	AND NOT GVL1.hwo_digitalAlarms[12].6	;	(*	DI:104	FIRE ALARM ACTVATED	*)
GVL1.Pwi_DigitalInputs[6].8	:= NOT w_im7IOStatus.8	AND NOT GVL1.hwo_digitalAlarms[12].6	;	(*	DI:105	AUTO PILOT FAIL ALARM	*)
GVL1.Pwi_DigitalInputs[6].9	:= NOT w_im7IOStatus.9	AND NOT GVL1.hwo_digitalAlarms[12].6	;	(*	DI:106	GAS DETECTION SYSTEM POWER FAIL	*)
GVL1.Pwi_DigitalInputs[6].10	:= NOT w_im7IOStatus.10	AND NOT GVL1.hwo_digitalAlarms[12].6	;	(*	DI:107	H2S ALARM ACTIVATED	*)
GVL1.Pwi_DigitalInputs[6].11	:= NOT w_im7IOStatus.11	AND NOT GVL1.hwo_digitalAlarms[12].6	;	(*	DI:108	LEL ALARM ACTIVATED	*)
GVL1.Pwi_DigitalInputs[6].12	:= NOT w_im7IOStatus.12	AND NOT GVL1.hwo_digitalAlarms[12].6	;	(*	DI:109	WH AREA REF. LEAKAGE ALARM 	*)
GVL1.Pwi_DigitalInputs[6].13	:= NOT w_im7IOStatus.13	AND NOT GVL1.hwo_digitalAlarms[12].6	;	(*	DI:110	PASSENGER AREA REF. LEAKAGE ALARM 	*)
GVL1.Pwi_DigitalInputs[6].14	:= NOT w_im7IOStatus.14	AND NOT GVL1.hwo_digitalAlarms[12].6	;	(*	DI:111	DEPTH BELOW KEEL LOWER THAN SET.P 	*)
GVL1.Pwi_DigitalInputs[6].15	:= NOT w_im7IOStatus.15	AND NOT GVL1.hwo_digitalAlarms[12].6	;	(*	DI:112	GMDSS COMMON ALRM	*)
//Digital input module1  MP- S3306: 16CH							
GVL1.Pwi_DigitalInputs[7].0	:= NOT w_im8IOstatus.0	AND NOT GVL1.hwo_digitalAlarms[12].7	;	(*	DI:113	PORT ME COMMON ALARM	*)
GVL1.Pwi_DigitalInputs[7].1	:= NOT w_im8IOstatus.1	AND NOT GVL1.hwo_digitalAlarms[12].7	;	(*	DI:114	STBD ME COMMON ALARM	*)
GVL1.Pwi_DigitalInputs[7].2	:= NOT w_im8IOstatus.2	AND NOT GVL1.hwo_digitalAlarms[12].7	;	(*	DI:115	CENTER ME COMMON ALARM	*)
GVL1.Pwi_DigitalInputs[7].3	:= NOT w_im8IOstatus.3	AND NOT GVL1.hwo_digitalAlarms[12].7	;	(*	DI:116	AUX COOLING PUMP-1 RUNNING	*)
GVL1.Pwi_DigitalInputs[7].4	:= NOT w_im8IOstatus.4	AND NOT GVL1.hwo_digitalAlarms[12].7	;	(*	DI:117	AUX COOLING PUMP-1 TRIP	*)
GVL1.Pwi_DigitalInputs[7].5	:= NOT w_im8IOstatus.5	AND NOT GVL1.hwo_digitalAlarms[12].7	;	(*	DI:118	FO PURIFIER COMMON ALRM	*)
GVL1.Pwi_DigitalInputs[7].6	:= NOT w_im8IOstatus.6	AND NOT GVL1.hwo_digitalAlarms[12].7	;	(*	DI:119	MSB: PREF. TRIP ALARM	*)
GVL1.Pwi_DigitalInputs[7].7	:= NOT w_im8IOstatus.7	AND NOT GVL1.hwo_digitalAlarms[12].7	;	(*	DI:120	MSB: 440V EARTH FAULT ALARM	*)
GVL1.Pwi_DigitalInputs[7].8	:= NOT w_im8IOstatus.8	AND NOT GVL1.hwo_digitalAlarms[12].7	;	(*	DI:121	MSB: 220V EARTH FAULT ALARM	*)
GVL1.Pwi_DigitalInputs[7].9	:= NOT w_im8IOstatus.9	AND NOT GVL1.hwo_digitalAlarms[12].7	;	(*	DI:122	MSB: 24VDC SUPPLY FAIL ALARM	*)
GVL1.Pwi_DigitalInputs[7].10	:= NOT w_im8IOstatus.10	AND NOT GVL1.hwo_digitalAlarms[12].7	;	(*	DI:123	MSB: ABNORMAL ALARM	*)
GVL1.Pwi_DigitalInputs[7].11	:= NOT w_im8IOstatus.11	AND NOT GVL1.hwo_digitalAlarms[12].7	;	(*	DI:124	AMS AC SUPPLY FAIL	*)
GVL1.Pwi_DigitalInputs[7].12	:= NOT w_im8IOstatus.12	AND NOT GVL1.hwo_digitalAlarms[12].7	;	(*	DI:125	AMS DC SUPPLY FAIL	*)
GVL1.Pwi_DigitalInputs[7].13	:= NOT w_im8IOstatus.13	AND NOT GVL1.hwo_digitalAlarms[12].7	;	(*	DI:126	ALRM MUTE AMS PANEL	*)
GVL1.Pwi_DigitalInputs[7].14	:= NOT w_im8IOstatus.14	AND NOT GVL1.hwo_digitalAlarms[12].7	;	(*	DI:127	SPARE	*)
GVL1.Pwi_DigitalInputs[7].15	:= NOT w_im8IOstatus.15	AND NOT GVL1.hwo_digitalAlarms[12].7	;	(*	DI:128	SPARE	*)
//Digital input module1  MP- S3306: 16CH							
GVL1.Pwi_DigitalInputs[8].0	:= NOT w_im9IOstatus.0	AND NOT GVL1.hwo_digitalAlarms[12].7	;	(*	DI:129	SPARE	*)
GVL1.Pwi_DigitalInputs[8].1	:= NOT w_im9IOstatus.1	AND NOT GVL1.hwo_digitalAlarms[12].7	;	(*	DI:130	SPARE	*)
GVL1.Pwi_DigitalInputs[8].2	:= NOT w_im9IOstatus.2	AND NOT GVL1.hwo_digitalAlarms[12].7	;	(*	DI:131	SPARE	*)
GVL1.Pwi_DigitalInputs[8].3	:= NOT w_im9IOstatus.3	AND NOT GVL1.hwo_digitalAlarms[12].7	;	(*	DI:132	SPARE	*)
GVL1.Pwi_DigitalInputs[8].4	:= NOT w_im9IOstatus.4	AND NOT GVL1.hwo_digitalAlarms[12].7	;	(*	DI:133	SPARE	*)
GVL1.Pwi_DigitalInputs[8].5	:= NOT w_im9IOstatus.5	AND NOT GVL1.hwo_digitalAlarms[12].7	;	(*	DI:134	SPARE	*)
GVL1.Pwi_DigitalInputs[8].6	:= NOT w_im9IOstatus.6	AND NOT GVL1.hwo_digitalAlarms[12].7	;	(*	DI:135	SPARE	*)
GVL1.Pwi_DigitalInputs[8].7	:= NOT w_im9IOstatus.7	AND NOT GVL1.hwo_digitalAlarms[12].7	;	(*	DI:136	SPARE	*)
GVL1.Pwi_DigitalInputs[8].8	:= NOT w_im9IOstatus.8	AND NOT GVL1.hwo_digitalAlarms[12].7	;	(*	DI:137	SPARE	*)
GVL1.Pwi_DigitalInputs[8].9	:= NOT w_im9IOstatus.9	AND NOT GVL1.hwo_digitalAlarms[12].7	;	(*	DI:138	SPARE	*)
GVL1.Pwi_DigitalInputs[8].10	:= NOT w_im9IOstatus.10	AND NOT GVL1.hwo_digitalAlarms[12].7	;	(*	DI:139	SPARE	*)
GVL1.Pwi_DigitalInputs[8].11	:= NOT w_im9IOstatus.11	AND NOT GVL1.hwo_digitalAlarms[12].7	;	(*	DI:140	SPARE	*)
GVL1.Pwi_DigitalInputs[8].12	:= NOT w_im9IOstatus.12	AND NOT GVL1.hwo_digitalAlarms[12].7	;	(*	DI:141	SPARE	*)
GVL1.Pwi_DigitalInputs[8].13	:= NOT w_im9IOstatus.13	AND NOT GVL1.hwo_digitalAlarms[12].7	;	(*	DI:142	SPARE	*)
GVL1.Pwi_DigitalInputs[8].14	:= NOT w_im9IOstatus.14	AND NOT GVL1.hwo_digitalAlarms[12].7	;	(*	DI:143	SPARE	*)
GVL1.Pwi_DigitalInputs[8].15	:= NOT w_im9IOstatus.15	AND NOT GVL1.hwo_digitalAlarms[12].7	;	(*	DI:144	SPARE	*)
//Digital I/O module MP- S3301: 8CH							
GVL1.Pwi_DigitalInputs[9].0	:=  w_iom1IStatus.0	AND NOT GVL1.hwo_digitalAlarms[12].8	;	(*	DI:145	SPARE	*)
GVL1.Pwi_DigitalInputs[9].1	:=  w_iom1IStatus.1	AND NOT GVL1.hwo_digitalAlarms[12].8	;	(*	DI:146	SPARE	*)
GVL1.Pwi_DigitalInputs[9].2	:=  w_iom1IStatus.2	AND NOT GVL1.hwo_digitalAlarms[12].8	;	(*	DI:147	SPARE	*)
GVL1.Pwi_DigitalInputs[9].3	:=  w_iom1IStatus.3	AND NOT GVL1.hwo_digitalAlarms[12].8	;	(*	DI:148	SPARE	*)
GVL1.Pwi_DigitalInputs[9].4	:=  w_iom1IStatus.4	AND NOT GVL1.hwo_digitalAlarms[12].8	;	(*	DI:149	SPARE	*)
GVL1.Pwi_DigitalInputs[9].5	:=  w_iom1IStatus.5	AND NOT GVL1.hwo_digitalAlarms[12].8	;	(*	DI:150	SPARE	*)
GVL1.Pwi_DigitalInputs[9].6	:=  w_iom1IStatus.6	AND NOT GVL1.hwo_digitalAlarms[12].8	;	(*	DI:151	SPARE	*)
GVL1.Pwi_DigitalInputs[9].7	:=  w_iom1IStatus.7	AND NOT GVL1.hwo_digitalAlarms[12].8	;	(*	DI:152	SPARE	*)




						
//Communication alarms - Soft channel: 16Ch					
GVL1.Pwi_DigitalInputs[12].0	 := NOT ton_blink11.Q	;	(*	JB1 DI MODULE COMMS: FAIL	*)
GVL1.Pwi_DigitalInputs[12].1	 := NOT ton_blink12.Q	;	(*	JB2 DI MODULE COMMS: FAIL	*)
GVL1.Pwi_DigitalInputs[12].2	 := NOT ton_blink13.Q	;	(*	JB3 DI MODULE COMMS: FAIL	*)
GVL1.Pwi_DigitalInputs[12].3	 := NOT ton_blink14.Q	;	(*	JB4 DI MODULE COMMS: FAIL	*)
GVL1.Pwi_DigitalInputs[12].4	 := NOT ton_blink15.Q	;	(*	JB5 DI MODULE COMMS: FAIL	*)
GVL1.Pwi_DigitalInputs[12].5	 := NOT ton_blink16.Q	;	(*	JB6 DI MODULE COMMS: FAIL	*)
GVL1.Pwi_DigitalInputs[12].6	 := NOT ton_blink17.Q	;	(*	WH DI MODULE COMMS: FAIL	*)
GVL1.Pwi_DigitalInputs[12].7	 := NOT ton_blink18.Q	;	(*	MP DI1 MODULE COMMS: FAIL	*)
GVL1.Pwi_DigitalInputs[12].8	 := NOT ton_blink19.Q	;	(*	MP DI2 MODULE COMMS: FAIL	*)
GVL1.Pwi_DigitalInputs[12].9	 := NOT ton_blink20.Q	;	(*	MP DIO MODULE COMMS: FAIL	*)
GVL1.Pwi_DigitalInputs[12].10	 := NOT ton_blink21.Q	;	(*	MP DO MODULE COMMS: FAIL	*)
GVL1.Pwi_DigitalInputs[12].11	 := NOT ton_blink22.Q	;	(*	MP AI MODULE COMMS: FAIL	*)
GVL1.Pwi_DigitalInputs[12].12	 := commCheck1.Lbo_ComErr1	; (*	ECR HMI COMMS: FAIL	*)			
GVL1.Pwi_DigitalInputs[12].13	 := commCheck1.Lbo_ComErr2	; (*	WH HMI COMMS: FAIL	*)		
GVL1.Pwi_DigitalInputs[12].14	 := commCheck1.Lbo_ComErr3	; (*	MESS HMI COMMS: FAIL	*)
GVL1.Pwi_DigitalInputs[12].15	 := 0	;			
	
	
			

(*Shore mode interlock for doors*)
lwi_interlocks[1].1 := GVL1.hxi_inhbit_doors;
lwi_interlocks[3].2 := GVL1.hxi_inhbit_doors;
lwi_interlocks[4].5  := GVL1.hxi_inhbit_doors;
lwi_interlocks[4].11  := GVL1.hxi_inhbit_doors;

//Digital IO module1 - S3303E: 8Ch		
w_iom1OStatus.0	 := NOT GVL1.pwo_digitalOutputs[0].0 	;	
w_iom1OStatus.1	 := NOT GVL1.pwo_digitalOutputs[0].1	;	
w_iom1OStatus.2	 := NOT GVL1.pwo_digitalOutputs[0].2	;	
w_iom1OStatus.3	 := NOT GVL1.pwo_digitalOutputs[0].3	;	
w_iom1OStatus.4	 := NOT GVL1.pwo_digitalOutputs[0].4	;	
w_iom1OStatus.5	 := NOT GVL1.pwo_digitalOutputs[0].5	;	



//Digital output module1 - S3303E: 16Ch	
poweron_ton(IN:=TRUE , PT:=T#10S , Q=> , ET=> );	
w_om1IOStatus.0	 := comAlarm.LDo_Accoustic1 AND poweron_ton.Q;	(*	VISUAL & AUDIO ALARM BUZZER ENG: ROOM	*)
w_om1IOStatus.1	 := comAlarm.LDo_Accoustic1 AND poweron_ton.Q;	(*	VISUAL & AUDIO ALARM BUZZER GEN: ROOM	*)
w_om1IOStatus.2	 := comAlarm.LDo_Accoustic1 AND poweron_ton.Q;	(*	VISUAL & AUDIO ALARM BUZZER PUMP ROOM	*)
w_om1IOStatus.3	 := comAlarm2.LDo_Accoustic1 AND poweron_ton.Q;		(*	BUZZER WITH IND MESS ROOM	*)
w_om1IOStatus.4	 := comAlarm1.LDo_Accoustic1 AND poweron_ton.Q;	(*	BUZZER WITH IND WHEEL HOUSE	*)

w_om1IOStatus.5	 := GVL1.pwo_digitalOutputs[1].5	;	(*	GREY WATER TANK LOW AUTO STOP GREY WATER PUMP PUMP	*)
IF GVL1.hwo_analogAlm[3].1 AND NOT GVL1.hwi_override.0 
THEN GVL1.pwo_digitalOutputs[1].5:= 1; ELSE GVL1.pwo_digitalOutputs[1].5:=0;	END_IF

w_om1IOStatus.6	 := GVL1.pwo_digitalOutputs[1].6	;	(*	FUEL TANK HIGH AUTO STOP FO PUMP	*)
IF (GVL1.hwo_analogAlm[4].2 AND NOT GVL1.hwi_override.1) OR (GVL1.hwo_analogAlm[5].2 AND NOT GVL1.hwi_override.2)
OR (GVL1.hwo_analogAlm[6].2 AND NOT GVL1.hwi_override.3) OR (GVL1.hwo_analogAlm[11].2 AND NOT GVL1.hwi_override.4)
OR (GVL1.hwo_analogAlm[12].2 AND NOT GVL1.hwi_override.5) OR (GVL1.hwo_analogAlm[13].2 AND NOT GVL1.hwi_override.6)
(*OR (GVL1.hwo_analogAlm[10].2 AND NOT GVL1.hwi_override.7)	*)
THEN GVL1.pwo_digitalOutputs[1].6:= 1; ELSE GVL1.pwo_digitalOutputs[1].6:=0;	END_IF

w_om1IOStatus.7	 := GVL1.pwo_digitalOutputs[1].7	;	(*	SLOPE TANK LOW AUTO STOP SLUDGE PUMP *)
IF GVL1.hwo_analogAlm[10].1 AND NOT GVL1.hwi_override.8 THEN GVL1.pwo_digitalOutputs[1].7:= 1; ELSE GVL1.pwo_digitalOutputs[1].7:=0;	END_IF

w_om1IOStatus.8:= GVL1.pwo_digitalOutputs[1].8	;(*	BT LOW OIL LEVEL / HIGH TEMP OUTPUT = engine sd	*)
ton_enginesd(IN:= GVL1.hwo_digitalAlarms[1].8 AND NOT overide_out, PT:= T#30S , Q=> , ET=> GVL1.enginesd_cd);
IF GVL1.hwo_digitalAlarms[1].8 AND (GVL1.hxi_enginesd_overide OR overide_out) THEN overide_out:=1 ;ELSE overide_out:=0; END_IF
IF (GVL1.hwo_digitalAlarms[1].8 OR GVL1.hwo_digitalAlarms[1].9) AND 
(GVL1.hxi_enginesd_accept OR GVL1.pwo_digitalOutputs[1].8 OR ton_enginesd.Q)
THEN GVL1.pwo_digitalOutputs[1].8:=1; ELSE GVL1.pwo_digitalOutputs[1].8:=0; END_IF

w_om1IOStatus.9	 := GVL1.pwo_digitalOutputs[1].9	;	(*	FODS HIGH AUTO STOP TO FO PURIFIER 	*)
IF (GVL1.hwo_analogAlm[8].2 AND NOT GVL1.hwi_override.9) OR (GVL1.hwo_analogAlm[9].2 AND NOT GVL1.hwi_override.10)
THEN GVL1.pwo_digitalOutputs[1].9:= 1; ELSE GVL1.pwo_digitalOutputs[1].9:=0;	END_IF

w_om1IOStatus.10:= GVL1.pwo_digitalOutputs[1].10	;	(*	FODS HIGH AUTO STOP TO FO PURIFIER 	*)
IF (GVL1.hwo_analogAlm[8].2 AND NOT GVL1.hwi_override.9) OR (GVL1.hwo_analogAlm[9].2 AND NOT GVL1.hwi_override.10)
THEN GVL1.pwo_digitalOutputs[1].10:= 1; ELSE GVL1.pwo_digitalOutputs[1].10:=0;	END_IF

w_om1IOStatus.11 := GVL1.pwo_digitalOutputs[1].11	;	(*	SPARE	*)
w_om1IOStatus.12 := GVL1.pwo_digitalOutputs[1].12	;	(*	SPARE	*)
w_om1IOStatus.13 := GVL1.pwo_digitalOutputs[1].13	;	(*	SPARE	*)
w_om1IOStatus.14 := GVL1.pwo_digitalOutputs[1].14	;	(*	SPARE	*)
w_om1IOStatus.15 := GVL1.pwo_digitalOutputs[1].15	;	(*	SPARE	*)



//Analog input module1 - S3103: 12Ch					
IF NOT GVL1.hwo_digitalAlarms[12].11 THEN					
GVL1.pwi_analogInput[0]	:= w_aim1ch1	;	(*	AI:01-FRESH WATER TANK 1C	*)
GVL1.pwi_analogInput[1]	:= w_aim1ch2	;	(*	AI:02-FRESH WATER TANK 2C	*)
GVL1.pwi_analogInput[2]	:= w_aim1ch3	;	(*	AI:03-BLACK WATER TANK	*)
GVL1.pwi_analogInput[3]	:= w_aim1ch4	;	(*	AI:04-GREY WATER TANK 	*)
GVL1.pwi_analogInput[4]	:= w_aim1ch5	;	(*	AI:05-FUEL OIL TANK PORT 1P	*)
GVL1.pwi_analogInput[5]	:= w_aim1ch6	;	(*	AI:06-FUEL OIL TANK STBD 1S	*)
GVL1.pwi_analogInput[6]	:= w_aim1ch7	;	(*	AI:07-FUEL OIL TANK PORT 3C	*)
GVL1.pwi_analogInput[7]	:= w_aim1ch8	;	(*	AI:08-BILGE HOLDING TANK	*)
GVL1.pwi_analogInput[8]	:= w_aim1ch9	;	(*	AI:09-FODS TANK PORT	*)
GVL1.pwi_analogInput[9]	:= w_aim1ch10	;	(*	AI:10-FODS TANK STDB	*)
GVL1.pwi_analogInput[10]	:= w_aim1ch11	;	(*	AI:11-SLOPE TANK 	*)
GVL1.pwi_analogInput[11]	:= w_aim1ch12	;	(*	AI:12-FUEL OIL TANK PORT 2C	*)
GVL1.pwi_analogInput[12]	:= w_aim1ch13	;	(*	AI:13-FUEL OIL TANK PORT 4P	*)
GVL1.pwi_analogInput[13]	:= w_aim1ch14	;	(*	AI:14-FUEL OIL TANK STBD 4S	*)
GVL1.pwi_analogInput[14]	:= w_aim1ch15	;	(*	SPARE	*)
GVL1.pwi_analogInput[15]	:= w_aim1ch16	;	(*	SPARE	*)

ELSE					
GVL1.pwi_analogInput[0]	:= 0;
GVL1.pwi_analogInput[1]	:= 0;
GVL1.pwi_analogInput[2]	:= 0;
GVL1.pwi_analogInput[3]	:= 0;
GVL1.pwi_analogInput[4]	:= 0;
GVL1.pwi_analogInput[5]	:= 0;
GVL1.pwi_analogInput[6]	:= 0;
GVL1.pwi_analogInput[7]	:= 0;
GVL1.pwi_analogInput[8]	:= 0;
GVL1.pwi_analogInput[9]	:= 0;
GVL1.pwi_analogInput[10]	:= 0;
GVL1.pwi_analogInput[11]	:= 0;
GVL1.pwi_analogInput[12]	:= 0;
GVL1.pwi_analogInput[13]	:= 0;
GVL1.pwi_analogInput[14]	:= 0;
GVL1.pwi_analogInput[15]	:= 0;
	
END_IF
END_ACTION

ACTION digitalProcessing:
(*Alarm/Event group 0*)
aeGroup0(
	wi_input:= GVL1.pwi_digitalInputs[0], 
	wi_set:= GVL1.hwi_digAlarmSet[0], 
	wai_delay:= GVL1.hwi_digAlarmDelay0, 
	wi_inhibit:= GVL1.hwi_digAlarmInh[0],
	wi_inhibitJm:= , 
	wi_interlock:= lwi_interlocks[0], 
	wi_alarmEvent:= GVL1.hwi_digAlarmOrEvent[0], 
	xi_reset:= lx_refresh, 
	xi_ack:= lx_ack, 
	wo_alarm=> GVL1.hwo_digitalAlarms[0], 
	wo_event=> GVL1.hwo_digitalEvents[0], 
	wo_alarmLa=> GVL1.hwo_digitalAlarmsp[0], 
	xo_buzzer=> lwo_dialmBuzzer.0, 
	xo_ind=> lwo_dialmInd.0, 
	xo_indLa=> ,
	wo_inhTot=>);
(*Alarm/Event group 1*)
aeGroup1(
	wi_input:= GVL1.pwi_digitalInputs[1], 
	wi_set:= GVL1.hwi_digAlarmSet[1], 
	wai_delay:= GVL1.hwi_digAlarmDelay1, 
	wi_inhibit:= GVL1.hwi_digAlarmInh[1],
	wi_inhibitJm:= , 
	wi_interlock:= lwi_interlocks[1], 
	wi_alarmEvent:= GVL1.hwi_digAlarmOrEvent[1], 
	xi_reset:= lx_refresh, 
	xi_ack:= lx_ack, 
	wo_alarm=> GVL1.hwo_digitalAlarms[1], 
	wo_event=> GVL1.hwo_digitalEvents[1], 
	wo_alarmLa=> GVL1.hwo_digitalAlarmsp[1], 
	xo_buzzer=> lwo_dialmBuzzer.1, 
	xo_ind=> lwo_dialmInd.1, 
	xo_indLa=> ,
	wo_inhTot=>);
(*Alarm/Event group 2*)
aeGroup2(
	wi_input:= GVL1.pwi_digitalInputs[2], 
	wi_set:= GVL1.hwi_digAlarmSet[2], 
	wai_delay:= GVL1.hwi_digAlarmDelay2, 
	wi_inhibit:= GVL1.hwi_digAlarmInh[2],
	wi_inhibitJm:= , 
	wi_interlock:= lwi_interlocks[2], 
	wi_alarmEvent:= GVL1.hwi_digAlarmOrEvent[2], 
	xi_reset:= lx_refresh, 
	xi_ack:= lx_ack, 
	wo_alarm=> GVL1.hwo_digitalAlarms[2], 
	wo_event=> GVL1.hwo_digitalEvents[2], 
	wo_alarmLa=> GVL1.hwo_digitalAlarmsp[2], 
	xo_buzzer=> lwo_dialmBuzzer.2, 
	xo_ind=> lwo_dialmInd.2, 
	xo_indLa=> ,
	wo_inhTot=>);
(*Alarm/Event group 3*)
aeGroup3(
	wi_input:= GVL1.pwi_digitalInputs[3], 
	wi_set:= GVL1.hwi_digAlarmSet[3], 
	wai_delay:= GVL1.hwi_digAlarmDelay3, 
	wi_inhibit:= GVL1.hwi_digAlarmInh[3],
	wi_inhibitJm:= , 
	wi_interlock:= lwi_interlocks[3], 
	wi_alarmEvent:= GVL1.hwi_digAlarmOrEvent[3], 
	xi_reset:= lx_refresh, 
	xi_ack:= lx_ack, 
	wo_alarm=> GVL1.hwo_digitalAlarms[3], 
	wo_event=> GVL1.hwo_digitalEvents[3], 
	wo_alarmLa=> GVL1.hwo_digitalAlarmsp[3], 
	xo_buzzer=> lwo_dialmBuzzer.3, 
	xo_ind=> lwo_dialmInd.3, 
	xo_indLa=> ,
	wo_inhTot=>);	
(*Alarm/Event group 4*)
aeGroup4(
	wi_input:= GVL1.pwi_digitalInputs[4], 
	wi_set:= GVL1.hwi_digAlarmSet[4], 
	wai_delay:= GVL1.hwi_digAlarmDelay4, 
	wi_inhibit:= GVL1.hwi_digAlarmInh[4],
	wi_inhibitJm:= , 
	wi_interlock:= lwi_interlocks[4], 
	wi_alarmEvent:= GVL1.hwi_digAlarmOrEvent[4], 
	xi_reset:= lx_refresh, 
	xi_ack:= lx_ack, 
	wo_alarm=> GVL1.hwo_digitalAlarms[4], 
	wo_event=> GVL1.hwo_digitalEvents[4], 
	wo_alarmLa=> GVL1.hwo_digitalAlarmsp[4], 
	xo_buzzer=> lwo_dialmBuzzer.4, 
	xo_ind=> lwo_dialmInd.4, 
	xo_indLa=> ,
	wo_inhTot=>);
(*Alarm/Event group 5*)
aeGroup5(
	wi_input:= GVL1.pwi_digitalInputs[5], 
	wi_set:= GVL1.hwi_digAlarmSet[5], 
	wai_delay:= GVL1.hwi_digAlarmDelay5, 
	wi_inhibit:= GVL1.hwi_digAlarmInh[5],
	wi_inhibitJm:= , 
	wi_interlock:= lwi_interlocks[5], 
	wi_alarmEvent:= GVL1.hwi_digAlarmOrEvent[5], 
	xi_reset:= lx_refresh, 
	xi_ack:= lx_ack, 
	wo_alarm=> GVL1.hwo_digitalAlarms[5], 
	wo_event=> GVL1.hwo_digitalEvents[5], 
	wo_alarmLa=> GVL1.hwo_digitalAlarmsp[5], 
	xo_buzzer=> lwo_dialmBuzzer.5, 
	xo_ind=> lwo_dialmInd.5, 
	xo_indLa=> ,
	wo_inhTot=>);
(*Alarm/Event group 6*)
aeGroup6(
	wi_input:= GVL1.pwi_digitalInputs[6], 
	wi_set:= GVL1.hwi_digAlarmSet[6], 
	wai_delay:= GVL1.hwi_digAlarmDelay6, 
	wi_inhibit:= GVL1.hwi_digAlarmInh[6],
	wi_inhibitJm:= , 
	wi_interlock:= lwi_interlocks[6], 
	wi_alarmEvent:= GVL1.hwi_digAlarmOrEvent[6], 
	xi_reset:= lx_refresh, 
	xi_ack:= lx_ack, 
	wo_alarm=> GVL1.hwo_digitalAlarms[6], 
	wo_event=> GVL1.hwo_digitalEvents[6], 
	wo_alarmLa=> GVL1.hwo_digitalAlarmsp[6], 
	xo_buzzer=> lwo_dialmBuzzer.6, 
	xo_ind=> lwo_dialmInd.6, 
	xo_indLa=> ,
	wo_inhTot=>);
(*Alarm/Event group 7*)
aeGroup7(
	wi_input:= GVL1.pwi_digitalInputs[7], 
	wi_set:= GVL1.hwi_digAlarmSet[7], 
	wai_delay:= GVL1.hwi_digAlarmDelay7, 
	wi_inhibit:= GVL1.hwi_digAlarmInh[7],
	wi_inhibitJm:= , 
	wi_interlock:= lwi_interlocks[7], 
	wi_alarmEvent:= GVL1.hwi_digAlarmOrEvent[7], 
	xi_reset:= lx_refresh, 
	xi_ack:= lx_ack, 
	wo_alarm=> GVL1.hwo_digitalAlarms[7], 
	wo_event=> GVL1.hwo_digitalEvents[7], 
	wo_alarmLa=> GVL1.hwo_digitalAlarmsp[7], 
	xo_buzzer=> lwo_dialmBuzzer.7, 
	xo_ind=> lwo_dialmInd.7, 
	xo_indLa=> ,
	wo_inhTot=>);
(*Alarm/Event group 8*)
aeGroup8(
	wi_input:= GVL1.pwi_digitalInputs[8], 
	wi_set:= GVL1.hwi_digAlarmSet[8], 
	wai_delay:= GVL1.hwi_digAlarmDelay8, 
	wi_inhibit:= GVL1.hwi_digAlarmInh[8],
	wi_inhibitJm:= , 
	wi_interlock:= lwi_interlocks[8], 
	wi_alarmEvent:= GVL1.hwi_digAlarmOrEvent[8], 
	xi_reset:= lx_refresh, 
	xi_ack:= lx_ack, 
	wo_alarm=> GVL1.hwo_digitalAlarms[8], 
	wo_event=> GVL1.hwo_digitalEvents[8], 
	wo_alarmLa=> GVL1.hwo_digitalAlarmsp[8], 
	xo_buzzer=> lwo_dialmBuzzer.8, 
	xo_ind=> lwo_dialmInd.8, 
	xo_indLa=> ,
	wo_inhTot=>);
	
(*Alarm/Event group 9*)
aeGroup9(
	wi_input:= GVL1.pwi_digitalInputs[9], 
	wi_set:= GVL1.hwi_digAlarmSet[9], 
	wai_delay:= GVL1.hwi_digAlarmDelay9, 
	wi_inhibit:= GVL1.hwi_digAlarmInh[9],
	wi_inhibitJm:= , 
	wi_interlock:= lwi_interlocks[9], 
	wi_alarmEvent:= GVL1.hwi_digAlarmOrEvent[9], 
	xi_reset:= lx_refresh, 
	xi_ack:= lx_ack, 
	wo_alarm=> GVL1.hwo_digitalAlarms[9], 
	wo_event=> GVL1.hwo_digitalEvents[9], 
	wo_alarmLa=> GVL1.hwo_digitalAlarmsp[9], 
	xo_buzzer=> lwo_dialmBuzzer.9, 
	xo_ind=> lwo_dialmInd.9, 
	xo_indLa=> ,
	wo_inhTot=>);

(*Alarm/Event group 10*)
aeGroup10(
	wi_input:= GVL1.pwi_digitalInputs[10], 
	wi_set:= GVL1.hwi_digAlarmSet[10], 
	wai_delay:= GVL1.hwi_digAlarmDelay10, 
	wi_inhibit:= GVL1.hwi_digAlarmInh[10],
	wi_inhibitJm:= , 
	wi_interlock:= lwi_interlocks[10], 
	wi_alarmEvent:= GVL1.hwi_digAlarmOrEvent[10], 
	xi_reset:= lx_refresh, 
	xi_ack:= lx_ack, 
	wo_alarm=> GVL1.hwo_digitalAlarms[10], 
	wo_event=> GVL1.hwo_digitalEvents[10], 
	wo_alarmLa=> GVL1.hwo_digitalAlarmsp[10], 
	xo_buzzer=> lwo_dialmBuzzer.10, 
	xo_ind=> lwo_dialmInd.10, 
	xo_indLa=> ,
	wo_inhTot=>);	
	
(*Alarm/Event group 11*)
aeGroup11(
	wi_input:= GVL1.pwi_digitalInputs[11], 
	wi_set:= GVL1.hwi_digAlarmSet[11], 
	wai_delay:= GVL1.hwi_digAlarmDelay11, 
	wi_inhibit:= GVL1.hwi_digAlarmInh[11],
	wi_inhibitJm:= , 
	wi_interlock:= lwi_interlocks[11], 
	wi_alarmEvent:= GVL1.hwi_digAlarmOrEvent[11], 
	xi_reset:= lx_refresh, 
	xi_ack:= lx_ack, 
	wo_alarm=> GVL1.hwo_digitalAlarms[11], 
	wo_event=> GVL1.hwo_digitalEvents[11], 
	wo_alarmLa=> GVL1.hwo_digitalAlarmsp[11], 
	xo_buzzer=> lwo_dialmBuzzer.11, 
	xo_ind=> lwo_dialmInd.11, 
	xo_indLa=> ,
	wo_inhTot=>);	
	
(*Alarm/Event group 12*)
aeGroup12(
	wi_input:= GVL1.pwi_digitalInputs[12], 
	wi_set:= GVL1.hwi_digAlarmSet[12], 
	wai_delay:= GVL1.hwi_digAlarmDelay12, 
	wi_inhibit:= GVL1.hwi_digAlarmInh[12],
	wi_inhibitJm:= , 
	wi_interlock:= lwi_interlocks[12], 
	wi_alarmEvent:= GVL1.hwi_digAlarmOrEvent[12], 
	xi_reset:= lx_refresh, 
	xi_ack:= lx_ack, 
	wo_alarm=> GVL1.hwo_digitalAlarms[12], 
	wo_event=> GVL1.hwo_digitalEvents[12], 
	wo_alarmLa=> GVL1.hwo_digitalAlarmsp[12], 
	xo_buzzer=> lwo_dialmBuzzer.12, 
	xo_ind=> lwo_dialmInd.12, 
	xo_indLa=> ,
	wo_inhTot=>);
END_ACTION

ACTION analogProcessing:
(*Tank monitor0 - FRESH WATER TANK 1C*)
tmGroup0(
	wi_sensorVal:= GVL1.pwi_analogInput[0], 
	wi_samplingIn:= GVL1.hwi_ch0X, 
	wi_samplingOut:= GVL1.hwi_ch0Y, 
	wi_chPara:= GVL1.hwi_chPara[0],
	wi_chParaJm:= , 
	xi_comErr:= GVL1.hwo_digitalAlarms[9].10, 
	xi_ack:= lx_ack, 
	ro_pressOut=> GVL1.hro_ch0OutVal[0], 
	ro_htOut=> GVL1.hro_ch0OutVal[1], 
	ro_volOut=> GVL1.hro_ch0OutVal[2], 
	ro_perOut=> GVL1.hro_ch0OutVal[3], 
	ro_curOut=> GVL1.hro_ch0OutVal[4], 
	wo_alarmOut=> GVL1.hwo_analogAlm[0], 
	wo_alarmOutp=> GVL1.hwo_analogAlmP[0], 
	xo_buzPulse=> lwo_aialmBuzzer.0, 
	xo_ind=> lwo_aialmInd.0, 
	wo_alarmMsg=> GVL1.hwo_almMsg[0],
	wo_inhTot=> , 
	ri_chSP:= GVL1.hri_chSP_Ch0);
	
(*Tank monitor1 - FRESH WATER TANK 2C*)
tmGroup1(
	wi_sensorVal:= GVL1.pwi_analogInput[1], 
	wi_samplingIn:= GVL1.hwi_ch1X, 
	wi_samplingOut:= GVL1.hwi_ch1Y, 
	wi_chPara:= GVL1.hwi_chPara[1],
	wi_chParaJm:= , 
	xi_comErr:= GVL1.hwo_digitalAlarms[9].10, 
	xi_ack:= lx_ack, 
	ro_pressOut=> GVL1.hro_ch1OutVal[0], 
	ro_htOut=> GVL1.hro_ch1OutVal[1], 
	ro_volOut=> GVL1.hro_ch1OutVal[2], 
	ro_perOut=> GVL1.hro_ch1OutVal[3], 
	ro_curOut=> GVL1.hro_ch1OutVal[4], 
	wo_alarmOut=> GVL1.hwo_analogAlm[1], 
	wo_alarmOutp=> GVL1.hwo_analogAlmP[1], 
	xo_buzPulse=> lwo_aialmBuzzer.1, 
	xo_ind=> lwo_aialmInd.1, 
	wo_alarmMsg=> GVL1.hwo_almMsg[1],
	wo_inhTot=> , 
	ri_chSP:= GVL1.hri_chSP_Ch1);
	
(*Tank monitor2 - BLACK WATER TANK*)
tmGroup2(
	wi_sensorVal:= GVL1.pwi_analogInput[2], 
	wi_samplingIn:= GVL1.hwi_ch2X, 
	wi_samplingOut:= GVL1.hwi_ch2Y, 
	wi_chPara:= GVL1.hwi_chPara[2],
	wi_chParaJm:= , 
	xi_comErr:= GVL1.hwo_digitalAlarms[9].10, 
	xi_ack:= lx_ack, 
	ro_pressOut=> GVL1.hro_ch2OutVal[0], 
	ro_htOut=> GVL1.hro_ch2OutVal[1], 
	ro_volOut=> GVL1.hro_ch2OutVal[2], 
	ro_perOut=> GVL1.hro_ch2OutVal[3], 
	ro_curOut=> GVL1.hro_ch2OutVal[4], 
	wo_alarmOut=> GVL1.hwo_analogAlm[2], 
	wo_alarmOutp=> GVL1.hwo_analogAlmP[2], 
	xo_buzPulse=> lwo_aialmBuzzer.2, 
	xo_ind=> lwo_aialmInd.2, 
	wo_alarmMsg=> GVL1.hwo_almMsg[2],
	wo_inhTot=> , 
	ri_chSP:= GVL1.hri_chSP_Ch2);
	
(*Tank monitor3 - GREY WATER TANK *)
tmGroup3(
	wi_sensorVal:= GVL1.pwi_analogInput[3], 
	wi_samplingIn:= GVL1.hwi_Ch3X, 
	wi_samplingOut:= GVL1.hwi_Ch3Y, 
	wi_chPara:= GVL1.hwi_chPara[3],
	wi_chParaJm:= , 
	xi_comErr:= GVL1.hwo_digitalAlarms[9].10, 
	xi_ack:= lx_ack, 
	ro_pressOut=> GVL1.hro_Ch3OutVal[0], 
	ro_htOut=> GVL1.hro_Ch3OutVal[1], 
	ro_volOut=> GVL1.hro_Ch3OutVal[2], 
	ro_perOut=> GVL1.hro_Ch3OutVal[3], 
	ro_curOut=> GVL1.hro_Ch3OutVal[4], 
	wo_alarmOut=> GVL1.hwo_analogAlm[3], 
	wo_alarmOutp=> GVL1.hwo_analogAlmP[3], 
	xo_buzPulse=> lwo_aialmBuzzer.3, 
	xo_ind=> lwo_aialmInd.3, 
	wo_alarmMsg=> GVL1.hwo_almMsg[3],
	wo_inhTot=> , 
	ri_chSP:= GVL1.hri_chSP_Ch3);	

(*Tank monitor4 - FUEL OIL TANK PORT 1P*)
tmGroup4(
	wi_sensorVal:= GVL1.pwi_analogInput[4], 
	wi_samplingIn:= GVL1.hwi_Ch4X, 
	wi_samplingOut:= GVL1.hwi_Ch4Y, 
	wi_chPara:= GVL1.hwi_chPara[4],
	wi_chParaJm:= , 
	xi_comErr:= GVL1.hwo_digitalAlarms[9].10, 
	xi_ack:= lx_ack, 
	ro_pressOut=> GVL1.hro_ch4OutVal[0], 
	ro_htOut=> GVL1.hro_Ch4OutVal[1], 
	ro_volOut=> GVL1.hro_Ch4OutVal[2], 
	ro_perOut=> GVL1.hro_Ch4OutVal[3], 
	ro_curOut=> GVL1.hro_Ch4OutVal[4], 
	wo_alarmOut=> GVL1.hwo_analogAlm[4], 
	wo_alarmOutp=> GVL1.hwo_analogAlmP[4], 
	xo_buzPulse=> lwo_aialmBuzzer.4, 
	xo_ind=> lwo_aialmInd.4, 
	wo_alarmMsg=> GVL1.hwo_almMsg[4],
	wo_inhTot=> , 
	ri_chSP:= GVL1.hri_chSP_Ch4);

(*Tank monitor5 - FUEL OIL TANK STBD 1S*)
tmGroup5(
	wi_sensorVal:= GVL1.pwi_analogInput[5], 
	wi_samplingIn:= GVL1.hwi_Ch5X, 
	wi_samplingOut:= GVL1.hwi_Ch5Y, 
	wi_chPara:= GVL1.hwi_chPara[5],
	wi_chParaJm:= , 
	xi_comErr:= GVL1.hwo_digitalAlarms[9].10, 
	xi_ack:= lx_ack, 
	ro_pressOut=> GVL1.hro_ch5OutVal[0], 
	ro_htOut=> GVL1.hro_Ch5OutVal[1], 
	ro_volOut=> GVL1.hro_Ch5OutVal[2], 
	ro_perOut=> GVL1.hro_Ch5OutVal[3], 
	ro_curOut=> GVL1.hro_Ch5OutVal[4], 
	wo_alarmOut=> GVL1.hwo_analogAlm[5], 
	wo_alarmOutp=> GVL1.hwo_analogAlmP[5], 
	xo_buzPulse=> lwo_aialmBuzzer.5, 
	xo_ind=> lwo_aialmInd.5, 
	wo_alarmMsg=> GVL1.hwo_almMsg[5],
	wo_inhTot=> , 
	ri_chSP:= GVL1.hri_chSP_Ch5);
	

(*Tank monitor6 - FUEL OIL TANK PORT 3C*)
tmGroup6(
	wi_sensorVal:= GVL1.pwi_analogInput[6], 
	wi_samplingIn:= GVL1.hwi_Ch6X, 
	wi_samplingOut:= GVL1.hwi_Ch6Y, 
	wi_chPara:= GVL1.hwi_chPara[6],
	wi_chParaJm:= , 
	xi_comErr:= GVL1.hwo_digitalAlarms[9].10, 
	xi_ack:= lx_ack, 
	ro_pressOut=> GVL1.hro_ch6OutVal[0], 
	ro_htOut=> GVL1.hro_Ch6OutVal[1], 
	ro_volOut=> GVL1.hro_Ch6OutVal[2], 
	ro_perOut=> GVL1.hro_Ch6OutVal[3], 
	ro_curOut=> GVL1.hro_Ch6OutVal[4], 
	wo_alarmOut=> GVL1.hwo_analogAlm[6], 
	wo_alarmOutp=> GVL1.hwo_analogAlmP[6], 
	xo_buzPulse=> lwo_aialmBuzzer.6, 
	xo_ind=> lwo_aialmInd.6, 
	wo_alarmMsg=> GVL1.hwo_almMsg[6],
	wo_inhTot=> , 
	ri_chSP:= GVL1.hri_chSP_Ch6);	
	
(*Tank monitor7 - BILGE HOLDING TANK*)
tmGroup7(
	wi_sensorVal:= GVL1.pwi_analogInput[7], 
	wi_samplingIn:= GVL1.hwi_Ch7X, 
	wi_samplingOut:= GVL1.hwi_Ch7Y, 
	wi_chPara:= GVL1.hwi_chPara[7],
	wi_chParaJm:= , 
	xi_comErr:= GVL1.hwo_digitalAlarms[9].10, 
	xi_ack:= lx_ack, 
	ro_pressOut=> GVL1.hro_ch7OutVal[0], 
	ro_htOut=> GVL1.hro_Ch7OutVal[1], 
	ro_volOut=> GVL1.hro_Ch7OutVal[2], 
	ro_perOut=> GVL1.hro_Ch7OutVal[3], 
	ro_curOut=> GVL1.hro_Ch7OutVal[4], 
	wo_alarmOut=> GVL1.hwo_analogAlm[7], 
	wo_alarmOutp=> GVL1.hwo_analogAlmP[7], 
	xo_buzPulse=> lwo_aialmBuzzer.7, 
	xo_ind=> lwo_aialmInd.7, 
	wo_alarmMsg=> GVL1.hwo_almMsg[7],
	wo_inhTot=> , 
	ri_chSP:= GVL1.hri_chSP_Ch7);

(*Tank monitor8 - FODS TANK PORT*)
tmGroup8(
	wi_sensorVal:= GVL1.pwi_analogInput[8], 
	wi_samplingIn:= GVL1.hwi_Ch8X, 
	wi_samplingOut:= GVL1.hwi_Ch8Y, 
	wi_chPara:= GVL1.hwi_chPara[8],
	wi_chParaJm:= , 
	xi_comErr:= GVL1.hwo_digitalAlarms[9].10, 
	xi_ack:= lx_ack, 
	ro_pressOut=> GVL1.hro_ch8OutVal[0], 
	ro_htOut=> GVL1.hro_Ch8OutVal[1], 
	ro_volOut=> GVL1.hro_Ch8OutVal[2], 
	ro_perOut=> GVL1.hro_Ch8OutVal[3], 
	ro_curOut=> GVL1.hro_Ch8OutVal[4], 
	wo_alarmOut=> GVL1.hwo_analogAlm[8], 
	wo_alarmOutp=> GVL1.hwo_analogAlmP[8], 
	xo_buzPulse=> lwo_aialmBuzzer.8, 
	xo_ind=> lwo_aialmInd.8, 
	wo_alarmMsg=> GVL1.hwo_almMsg[8],
	wo_inhTot=> , 
	ri_chSP:= GVL1.hri_chSP_Ch8);
	
(*Tank monitor9 - FODS TANK STDB*)
tmGroup9(
	wi_sensorVal:= GVL1.pwi_analogInput[9], 
	wi_samplingIn:= GVL1.hwi_Ch9X, 
	wi_samplingOut:= GVL1.hwi_Ch9Y, 
	wi_chPara:= GVL1.hwi_chPara[9],
	wi_chParaJm:= , 
	xi_comErr:= GVL1.hwo_digitalAlarms[9].10, 
	xi_ack:= lx_ack, 
	ro_pressOut=> GVL1.hro_ch9OutVal[0], 
	ro_htOut=> GVL1.hro_Ch9OutVal[1], 
	ro_volOut=> GVL1.hro_Ch9OutVal[2], 
	ro_perOut=> GVL1.hro_Ch9OutVal[3], 
	ro_curOut=> GVL1.hro_Ch9OutVal[4], 
	wo_alarmOut=> GVL1.hwo_analogAlm[9], 
	wo_alarmOutp=> GVL1.hwo_analogAlmP[9], 
	xo_buzPulse=> lwo_aialmBuzzer.9, 
	xo_ind=> lwo_aialmInd.9, 
	wo_alarmMsg=> GVL1.hwo_almMsg[9],
	wo_inhTot=> , 
	ri_chSP:= GVL1.hri_chSP_Ch9);
	
(*Tank monitor10 - SLOPE TANK *)
tmGroup10(
	wi_sensorVal:= GVL1.pwi_analogInput[10], 
	wi_samplingIn:= GVL1.hwi_Ch10X, 
	wi_samplingOut:= GVL1.hwi_Ch10Y, 
	wi_chPara:= GVL1.hwi_chPara[10],
	wi_chParaJm:= , 
	xi_comErr:= GVL1.hwo_digitalAlarms[9].10, 
	xi_ack:= lx_ack, 
	ro_pressOut=> GVL1.hro_ch10OutVal[0], 
	ro_htOut=> GVL1.hro_Ch10OutVal[1], 
	ro_volOut=> GVL1.hro_Ch10OutVal[2], 
	ro_perOut=> GVL1.hro_Ch10OutVal[3], 
	ro_curOut=> GVL1.hro_Ch10OutVal[4], 
	wo_alarmOut=> GVL1.hwo_analogAlm[10], 
	wo_alarmOutp=> GVL1.hwo_analogAlmP[10], 
	xo_buzPulse=> lwo_aialmBuzzer.10, 
	xo_ind=> lwo_aialmInd.10, 
	wo_alarmMsg=> GVL1.hwo_almMsg[10],
	wo_inhTot=> , 
	ri_chSP:= GVL1.hri_chSP_Ch10);
	
(*Tank monitor11 - FUEL OIL TANK PORT 2C*)
tmGroup11(
	wi_sensorVal:= GVL1.pwi_analogInput[11], 
	wi_samplingIn:= GVL1.hwi_Ch11X, 
	wi_samplingOut:= GVL1.hwi_Ch11Y, 
	wi_chPara:= GVL1.hwi_chPara[11],
	wi_chParaJm:= , 
	xi_comErr:= GVL1.hwo_digitalAlarms[9].10, 
	xi_ack:= lx_ack, 
	ro_pressOut=> GVL1.hro_ch11OutVal[0], 
	ro_htOut=> GVL1.hro_Ch11OutVal[1], 
	ro_volOut=> GVL1.hro_Ch11OutVal[2], 
	ro_perOut=> GVL1.hro_Ch11OutVal[3], 
	ro_curOut=> GVL1.hro_Ch11OutVal[4], 
	wo_alarmOut=> GVL1.hwo_analogAlm[11], 
	wo_alarmOutp=> GVL1.hwo_analogAlmP[11], 
	xo_buzPulse=> lwo_aialmBuzzer.11, 
	xo_ind=> lwo_aialmInd.11, 
	wo_alarmMsg=> GVL1.hwo_almMsg[11],
	wo_inhTot=> , 
	ri_chSP:= GVL1.hri_chSP_Ch11);	
	
	(*Tank monitor12 - FUEL OIL TANK PORT 4P*)
tmGroup12(
	wi_sensorVal:= GVL1.pwi_analogInput[12], 
	wi_samplingIn:= GVL1.hwi_Ch12X, 
	wi_samplingOut:= GVL1.hwi_Ch12Y, 
	wi_chPara:= GVL1.hwi_chPara[12],
	wi_chParaJm:= , 
	xi_comErr:= GVL1.hwo_digitalAlarms[9].10, 
	xi_ack:= lx_ack, 
	ro_pressOut=> GVL1.hro_ch12OutVal[0], 
	ro_htOut=> GVL1.hro_Ch12OutVal[1], 
	ro_volOut=> GVL1.hro_Ch12OutVal[2], 
	ro_perOut=> GVL1.hro_Ch12OutVal[3], 
	ro_curOut=> GVL1.hro_Ch12OutVal[4], 
	wo_alarmOut=> GVL1.hwo_analogAlm[12], 
	wo_alarmOutp=> GVL1.hwo_analogAlmP[12], 
	xo_buzPulse=> lwo_aialmBuzzer.12, 
	xo_ind=> lwo_aialmInd.12, 
	wo_alarmMsg=> GVL1.hwo_almMsg[12],
	wo_inhTot=> , 
	ri_chSP:= GVL1.hri_chSP_Ch12);	

	(*Tank monitor13 - FUEL OIL TANK STBD 4S*)
tmGroup13(
	wi_sensorVal:= GVL1.pwi_analogInput[13], 
	wi_samplingIn:= GVL1.hwi_Ch13X, 
	wi_samplingOut:= GVL1.hwi_Ch13Y, 
	wi_chPara:= GVL1.hwi_chPara[13],
	wi_chParaJm:= , 
	xi_comErr:= GVL1.hwo_digitalAlarms[9].10, 
	xi_ack:= lx_ack, 
	ro_pressOut=> GVL1.hro_ch13OutVal[0], 
	ro_htOut=> GVL1.hro_Ch13OutVal[1], 
	ro_volOut=> GVL1.hro_Ch13OutVal[2], 
	ro_perOut=> GVL1.hro_Ch13OutVal[3], 
	ro_curOut=> GVL1.hro_Ch13OutVal[4], 
	wo_alarmOut=> GVL1.hwo_analogAlm[13], 
	wo_alarmOutp=> GVL1.hwo_analogAlmP[13], 
	xo_buzPulse=> lwo_aialmBuzzer.13, 
	xo_ind=> lwo_aialmInd.13, 
	wo_alarmMsg=> GVL1.hwo_almMsg[13],
	wo_inhTot=> , 
	ri_chSP:= GVL1.hri_chSP_Ch13);
	
(*Tank monitor14 - spare*)
tmGroup14(
	wi_sensorVal:= GVL1.pwi_analogInput[14], 
	wi_samplingIn:= GVL1.hwi_Ch14X, 
	wi_samplingOut:= GVL1.hwi_Ch14Y, 
	wi_chPara:= GVL1.hwi_chPara[14],
	wi_chParaJm:= , 
	xi_comErr:= GVL1.hwo_digitalAlarms[9].10, 
	xi_ack:= lx_ack, 
	ro_pressOut=> GVL1.hro_ch14OutVal[0], 
	ro_htOut=> GVL1.hro_Ch14OutVal[1], 
	ro_volOut=> GVL1.hro_Ch14OutVal[2], 
	ro_perOut=> GVL1.hro_Ch14OutVal[3], 
	ro_curOut=> GVL1.hro_Ch14OutVal[4], 
	wo_alarmOut=> GVL1.hwo_analogAlm[14], 
	wo_alarmOutp=> GVL1.hwo_analogAlmP[14], 
	xo_buzPulse=> lwo_aialmBuzzer.14, 
	xo_ind=> lwo_aialmInd.14, 
	wo_alarmMsg=> GVL1.hwo_almMsg[14],
	wo_inhTot=> , 
	ri_chSP:= GVL1.hri_chSP_Ch14);

(*Tank monitor15 - spare*)
tmGroup15(
	wi_sensorVal:= GVL1.pwi_analogInput[15], 
	wi_samplingIn:= GVL1.hwi_Ch15X, 
	wi_samplingOut:= GVL1.hwi_Ch15Y, 
	wi_chPara:= GVL1.hwi_chPara[15],
	wi_chParaJm:= , 
	xi_comErr:= GVL1.hwo_digitalAlarms[9].10, 
	xi_ack:= lx_ack, 
	ro_pressOut=> GVL1.hro_ch15OutVal[0], 
	ro_htOut=> GVL1.hro_Ch15OutVal[1], 
	ro_volOut=> GVL1.hro_Ch15OutVal[2], 
	ro_perOut=> GVL1.hro_Ch15OutVal[3], 
	ro_curOut=> GVL1.hro_Ch15OutVal[4], 
	wo_alarmOut=> GVL1.hwo_analogAlm[15], 
	wo_alarmOutp=> GVL1.hwo_analogAlmP[15], 
	xo_buzPulse=> lwo_aialmBuzzer.15, 
	xo_ind=> lwo_aialmInd.15, 
	wo_alarmMsg=> GVL1.hwo_almMsg[15],
	wo_inhTot=> , 
	ri_chSP:= GVL1.hri_chSP_Ch15);
END_ACTION

ACTION commReset:
x_im1Error := Modbus_Slave_im1.xError;
im1Errorcode := Modbus_Slave_im1.byModbusError;
//Modbus_Slave_im1.xAcknowledge := x_im1Ack;
(*
Modbus_Slave_im1.xReset := x_im1Reset OR x_mbReset;
Modbus_Slave_im2.xReset := x_im2Reset OR x_mbReset;
Modbus_Slave_im3.xReset := x_im3Reset OR x_mbReset;
Modbus_Slave_im4.xReset := x_im4Reset OR x_mbReset;
Modbus_Slave_im5.xReset := x_im5Reset OR x_mbReset;
Modbus_Slave_im6.xReset := x_im6Reset OR x_mbReset;
Modbus_Slave_im7.xReset := x_im7Reset OR x_mbReset;
Modbus_Slave_om1.xReset := x_om1Reset OR x_mbReset;
Modbus_Slave_aim1.xReset := x_aim1Reset OR x_mbReset;

(*Individual cyclic reset*)

ton_blink1(IN:= Modbus_Slave_im1.xError AND NOT x_im1Reset, PT:= T#1S, Q=> x_im1Reset, ET=> );
ton_blink2(IN:= Modbus_Slave_im2.xError AND NOT x_im2Reset, PT:= T#1S, Q=> x_im2Reset, ET=> );
ton_blink3(IN:= Modbus_Slave_im3.xError AND NOT x_im3Reset, PT:= T#1S, Q=> x_im3Reset, ET=> );
ton_blink4(IN:= Modbus_Slave_im4.xError AND NOT x_im4Reset, PT:= T#1S, Q=> x_im4Reset, ET=> );
ton_blink5(IN:= Modbus_Slave_im5.xError AND NOT x_im5Reset, PT:= T#1S, Q=> x_im5Reset, ET=> );
ton_blink6(IN:= Modbus_Slave_im6.xError AND NOT x_im6Reset, PT:= T#1S, Q=> x_im6Reset, ET=> );
ton_blink7(IN:= Modbus_Slave_im7.xError AND NOT x_im7Reset, PT:= T#1S, Q=> x_im7Reset, ET=> );
ton_blink8(IN:= Modbus_Slave_om1.xError AND NOT x_om1Reset, PT:= T#1S, Q=> x_om1Reset, ET=> );
ton_blink9(IN:= Modbus_Slave_aim1.xError AND NOT x_aim1Reset, PT:= T#1S, Q=> x_aim1Reset, ET=> );
*)
(*Common reset*)

ton_blink11(IN:= NOT Modbus_Slave_im1.xError, PT:= T#5S, Q=> , ET=> );
ton_blink12(IN:= NOT Modbus_Slave_im2.xError, PT:= T#5S, Q=> , ET=> );
ton_blink13(IN:= NOT Modbus_Slave_im3.xError, PT:= T#5S, Q=> , ET=> );
ton_blink14(IN:= NOT Modbus_Slave_im4.xError, PT:= T#5S, Q=> , ET=> );
ton_blink15(IN:= NOT Modbus_Slave_im5.xError, PT:= T#5S, Q=> , ET=> );
ton_blink16(IN:= NOT Modbus_Slave_im6.xError, PT:= T#5S, Q=> , ET=> );
ton_blink17(IN:= NOT Modbus_Slave_im7.xError, PT:= T#5S, Q=> , ET=> );
ton_blink18(IN:= NOT Modbus_Slave_im8.xError, PT:= T#5S, Q=> , ET=> );
ton_blink19(IN:= NOT Modbus_Slave_im9.xError, PT:= T#5S, Q=> , ET=> );
ton_blink20(IN:= NOT Modbus_Slave_iom1.xError, PT:= T#5S, Q=> , ET=> );
ton_blink21(IN:= NOT Modbus_Slave_om1.xError, PT:= T#5S, Q=> , ET=> );
ton_blink22(IN:= NOT Modbus_Slave_aim1.xError, PT:= T#5S, Q=> , ET=> );
(*Common reset*)
(*
tp_blink1(IN:= ton_blink11.Q, PT:= T#1S, Q=> , ET=> );
tp_blink2(IN:= ton_blink12.Q, PT:= T#1S, Q=> , ET=> );
tp_blink3(IN:= ton_blink13.Q, PT:= T#1S, Q=> , ET=> );
tp_blink4(IN:= ton_blink14.Q, PT:= T#1S, Q=> , ET=> );
tp_blink5(IN:= ton_blink15.Q, PT:= T#1S, Q=> , ET=> );
tp_blink6(IN:= ton_blink16.Q, PT:= T#1S, Q=> , ET=> );
tp_blink7(IN:= ton_blink17.Q, PT:= T#1S, Q=> , ET=> );
tp_blink8(IN:= ton_blink18.Q, PT:= T#1S, Q=> , ET=> );
tp_blink9(IN:= ton_blink19.Q, PT:= T#1S, Q=> , ET=> );

tp_blink11(IN:= NOT ton_blink11.Q, PT:= T#1S, Q=> , ET=> );
tp_blink12(IN:= NOT ton_blink12.Q, PT:= T#1S, Q=> , ET=> );
tp_blink13(IN:= NOT ton_blink13.Q, PT:= T#1S, Q=> , ET=> );
tp_blink14(IN:= NOT ton_blink14.Q, PT:= T#1S, Q=> , ET=> );
tp_blink15(IN:= NOT ton_blink15.Q, PT:= T#1S, Q=> , ET=> );
tp_blink16(IN:= NOT ton_blink16.Q, PT:= T#1S, Q=> , ET=> );
tp_blink17(IN:= NOT ton_blink17.Q, PT:= T#1S, Q=> , ET=> );
tp_blink18(IN:= NOT ton_blink18.Q, PT:= T#1S, Q=> , ET=> );
tp_blink19(IN:= NOT ton_blink19.Q, PT:= T#1S, Q=> , ET=> );

x_mbReset := tp_blink11.Q OR tp_blink12.Q OR tp_blink13.Q OR tp_blink14.Q OR tp_blink15.Q OR
tp_blink16.Q OR tp_blink17.Q OR tp_blink18.Q OR tp_blink19.Q OR
tp_blink1.Q OR tp_blink2.Q OR tp_blink3.Q OR tp_blink4.Q OR tp_blink5.Q OR
tp_blink6.Q OR tp_blink7.Q OR tp_blink8.Q OR tp_blink9.Q;
*)
END_ACTION

ACTION alarmOut:
lx_ack := GVL1.hxi_ack OR GVL1.hxi_ackEr ;
(*ER*)
buzzerSet1(
	Lwi_AlarmBuzzer:= lwo_dialmBuzzer, 
	Lwi_AlarmInd:= lwo_dialmInd, 
	LDi_Ack:= comAlarm.LDo_BuzStop, 
	LDo_Acoustic=> , 
	LDo_Visual=> );
buzzerSet2(
	Lwi_AlarmBuzzer:= lwo_aialmBuzzer, 
	Lwi_AlarmInd:= lwo_aialmInd, 
	LDi_Ack:= comAlarm.LDo_BuzStop, 
	LDo_Acoustic=> , 
	LDo_Visual=> );
	
comAlarm(
	LDi_Accoustic1:= buzzerSet1.LDo_Acoustic, 
	LDi_Accoustic2:= buzzerSet2.LDo_Acoustic, 
	LDi_Accoustic3:= , 
	LDi_Visual1:= buzzerSet1.LDo_Visual, 
	LDi_Visual2:= buzzerSet2.LDo_Visual, 
	LDi_Visual3:= , 
	LDi_BuzStop1:= GVL1.hxi_silence OR GVL1.hxi_silenceEr OR GVL1.Pwi_DigitalInputs[7].13, 
	LDi_BuzStop2:= GVL1.hxi_ack OR GVL1.hxi_ackEr, 
	LDi_BuzStop3:= , 
	LDi_BuzStop4:= , 
	LDi_Ack1:= GVL1.hxi_ack, 
	LDi_Ack2:= , 
	LDi_Ack3:= , 
	LDi_Ack4:= , 
	LDo_Accoustic1=> , 
	LDo_Accoustic2=> , 
	LDo_Visual1=> , 
	LDo_Visual2=> , 
	LDo_BuzStop=> , 
	LDo_Ack=> );
	
(*WH*)
buzzerSet3(
	Lwi_AlarmBuzzer:= lwo_dialmBuzzer, 
	Lwi_AlarmInd:= lwo_dialmInd, 
	LDi_Ack:= comAlarm1.LDo_BuzStop, 
	LDo_Acoustic=> , 
	LDo_Visual=> );
buzzerSet4(
	Lwi_AlarmBuzzer:= lwo_aialmBuzzer, 
	Lwi_AlarmInd:= lwo_aialmInd, 
	LDi_Ack:= comAlarm1.LDo_BuzStop, 
	LDo_Acoustic=> , 
	LDo_Visual=> );
	
comAlarm1(
	LDi_Accoustic1:= buzzerSet3.LDo_Acoustic, 
	LDi_Accoustic2:= buzzerSet4.LDo_Acoustic, 
	LDi_Accoustic3:= , 
	LDi_Visual1:= buzzerSet3.LDo_Visual, 
	LDi_Visual2:= buzzerSet4.LDo_Visual, 
	LDi_Visual3:= , 
	LDi_BuzStop1:= GVL1.hxi_silence  OR GVL1.hxi_silenceEr OR GVL1.hxi_silenceWh OR GVL1.Pwi_DigitalInputs[7].13 OR GVL1.Pwi_DigitalInputs[6].0 , 
	LDi_BuzStop2:= GVL1.hxi_ack OR GVL1.hxi_ackWh OR GVL1.hxi_ackEr, 
	LDi_BuzStop3:= , 
	LDi_BuzStop4:= , 
	LDi_Ack1:= GVL1.hxi_ack, 
	LDi_Ack2:= GVL1.hxi_ackWh, 
	LDi_Ack3:= GVL1.hxi_ackEr, 
	LDi_Ack4:= , 
	LDo_Accoustic1=> , 
	LDo_Accoustic2=> , 
	LDo_Visual1=> , 
	LDo_Visual2=> , 
	LDo_BuzStop=> , 
	LDo_Ack=> GVL1.hxi_ackWhout);	

(*MESS*)
buzzerSet5(
	Lwi_AlarmBuzzer:= lwo_dialmBuzzer, 
	Lwi_AlarmInd:= lwo_dialmInd, 
	LDi_Ack:= comAlarm2.LDo_BuzStop, 
	LDo_Acoustic=> , 
	LDo_Visual=> );
buzzerSet6(
	Lwi_AlarmBuzzer:= lwo_aialmBuzzer, 
	Lwi_AlarmInd:= lwo_aialmInd, 
	LDi_Ack:= comAlarm2.LDo_BuzStop, 
	LDo_Acoustic=> , 
	LDo_Visual=> );
	
comAlarm2(
	LDi_Accoustic1:= buzzerSet5.LDo_Acoustic, 
	LDi_Accoustic2:= buzzerSet6.LDo_Acoustic, 
	LDi_Accoustic3:= , 
	LDi_Visual1:= buzzerSet5.LDo_Visual, 
	LDi_Visual2:= buzzerSet6.LDo_Visual, 
	LDi_Visual3:= , 
	LDi_BuzStop1:= GVL1.hxi_silence  OR GVL1.hxi_silenceEr OR GVL1.hxi_silenceMess OR GVL1.Pwi_DigitalInputs[7].13  , 
	LDi_BuzStop2:= GVL1.hxi_ack OR GVL1.hxi_ackMess OR GVL1.hxi_ackEr, 
	LDi_BuzStop3:= , 
	LDi_BuzStop4:= , 
	LDi_Ack1:= GVL1.hxi_ack, 
	LDi_Ack2:= GVL1.hxi_ackMess, 
	LDi_Ack3:= GVL1.hxi_ackEr, 
	LDi_Ack4:= , 
	LDo_Accoustic1=> , 
	LDo_Accoustic2=> , 
	LDo_Visual1=> , 
	LDo_Visual2=> , 
	LDo_BuzStop=> , 
	LDo_Ack=> GVL1.hxi_ackMessout );


	
GVL1.hxo_alarmInd := comAlarm.LDo_Accoustic1;
GVL1.hxo_alarmIndwh := comAlarm1.LDo_Accoustic1;
GVL1.hxo_alarmIndMess := comAlarm2.LDo_Accoustic1;

commCheck1(
	Lbi_Enable:= TRUE, 
	Lbi_Resp1:= GVL1.Hbi_HMI1Resp, 
	Lbi_Resp2:= GVL1.Hbi_HMI2Resp, 
	Lbi_Resp3:= GVL1.Hbi_HMI3Resp, 
	Lbi_Resp4:= , 
	Lbo_Request=> GVL1.Hbo_HMITest, 
	Lbo_ComErr1=> , 
	Lbo_ComErr2=> , 
	Lbo_ComErr3=> , 
	Lbo_ComErr4=> );
END_ACTION

ACTION alarmInh:
GVL1.hwo_inhibited := aeGroup0.wo_inhTot + aeGroup1.wo_inhTot + aeGroup2.wo_inhTot + aeGroup3.wo_inhTot
+ aeGroup4.wo_inhTot + aeGroup5.wo_inhTot + aeGroup6.wo_inhTot + aeGroup7.wo_inhTot + aeGroup8.wo_inhTot
+ aeGroup9.wo_inhTot (*+ aeGroup10.wo_inhTot + aeGroup11.wo_inhTot*) + aeGroup12.wo_inhTot + tmGroup0.wo_inhTot 
+ tmGroup1.wo_inhTot + tmGroup2.wo_inhTot + tmGroup3.wo_inhTot + tmGroup4.wo_inhTot + tmGroup5.wo_inhTot 
+ tmGroup6.wo_inhTot + tmGroup7.wo_inhTot + tmGroup8.wo_inhTot + tmGroup9.wo_inhTot + tmGroup10.wo_inhTot
+ tmGroup11.wo_inhTot + tmGroup12.wo_inhTot + tmGroup13.wo_inhTot (*+ tmGroup14.wo_inhTot + tmGroup15.wo_inhTot*);
 


GVL1.hxo_inhibited := GVL1.hwo_inhibited > 0 ;

aeGroup0.wi_inhibitJm.0	:=	NOT GVL1.hxi_alarmInh[0	];
aeGroup0.wi_inhibitJm.1	:=	NOT GVL1.hxi_alarmInh[1	];
aeGroup0.wi_inhibitJm.2	:=	NOT GVL1.hxi_alarmInh[2	];
aeGroup0.wi_inhibitJm.3	:=	NOT GVL1.hxi_alarmInh[3	];
aeGroup0.wi_inhibitJm.4	:=	NOT GVL1.hxi_alarmInh[4	];
aeGroup0.wi_inhibitJm.5	:=	NOT GVL1.hxi_alarmInh[5	];
aeGroup0.wi_inhibitJm.6	:=	NOT GVL1.hxi_alarmInh[6	];
aeGroup0.wi_inhibitJm.7	:=	NOT GVL1.hxi_alarmInh[7	];
aeGroup0.wi_inhibitJm.8	:=	NOT GVL1.hxi_alarmInh[8	];
aeGroup0.wi_inhibitJm.9	:=	NOT GVL1.hxi_alarmInh[9	];
aeGroup0.wi_inhibitJm.10	:=	NOT GVL1.hxi_alarmInh[10	];
aeGroup0.wi_inhibitJm.11	:=	NOT GVL1.hxi_alarmInh[11	];
aeGroup0.wi_inhibitJm.12	:=	NOT GVL1.hxi_alarmInh[12	];
aeGroup0.wi_inhibitJm.13	:=	NOT GVL1.hxi_alarmInh[13	];
aeGroup0.wi_inhibitJm.14	:=	NOT GVL1.hxi_alarmInh[14	];
aeGroup0.wi_inhibitJm.15	:=	NOT GVL1.hxi_alarmInh[15	];
			
aeGroup1.wi_inhibitJm.0	:=	NOT GVL1.hxi_alarmInh[16	];
aeGroup1.wi_inhibitJm.1	:=	NOT GVL1.hxi_alarmInh[17	];
aeGroup1.wi_inhibitJm.2	:=	NOT GVL1.hxi_alarmInh[18	];
aeGroup1.wi_inhibitJm.3	:=	NOT GVL1.hxi_alarmInh[19	];
aeGroup1.wi_inhibitJm.4	:=	NOT GVL1.hxi_alarmInh[20	];
aeGroup1.wi_inhibitJm.5	:=	NOT GVL1.hxi_alarmInh[21	];
aeGroup1.wi_inhibitJm.6	:=	NOT GVL1.hxi_alarmInh[22	];
aeGroup1.wi_inhibitJm.7	:=	NOT GVL1.hxi_alarmInh[23	];
aeGroup1.wi_inhibitJm.8	:=	NOT GVL1.hxi_alarmInh[24	];
aeGroup1.wi_inhibitJm.9	:=	NOT GVL1.hxi_alarmInh[25	];
aeGroup1.wi_inhibitJm.10	:=	NOT GVL1.hxi_alarmInh[26	];
aeGroup1.wi_inhibitJm.11	:=	NOT GVL1.hxi_alarmInh[27	];
aeGroup1.wi_inhibitJm.12	:=	NOT GVL1.hxi_alarmInh[28	];
aeGroup1.wi_inhibitJm.13	:=	NOT GVL1.hxi_alarmInh[29	];
aeGroup1.wi_inhibitJm.14	:=	NOT GVL1.hxi_alarmInh[30	];
aeGroup1.wi_inhibitJm.15	:=	NOT GVL1.hxi_alarmInh[31	];
			
aeGroup2.wi_inhibitJm.0	:=	NOT GVL1.hxi_alarmInh[32	];
aeGroup2.wi_inhibitJm.1	:=	NOT GVL1.hxi_alarmInh[33	];
aeGroup2.wi_inhibitJm.2	:=	NOT GVL1.hxi_alarmInh[34	];
aeGroup2.wi_inhibitJm.3	:=	NOT GVL1.hxi_alarmInh[35	];
aeGroup2.wi_inhibitJm.4	:=	NOT GVL1.hxi_alarmInh[36	];
aeGroup2.wi_inhibitJm.5	:=	NOT GVL1.hxi_alarmInh[37	];
aeGroup2.wi_inhibitJm.6	:=	NOT GVL1.hxi_alarmInh[38	];
aeGroup2.wi_inhibitJm.7	:=	NOT GVL1.hxi_alarmInh[39	];
aeGroup2.wi_inhibitJm.8	:=	NOT GVL1.hxi_alarmInh[40	];
aeGroup2.wi_inhibitJm.9	:=	NOT GVL1.hxi_alarmInh[41	];
aeGroup2.wi_inhibitJm.10	:=	NOT GVL1.hxi_alarmInh[42	];
aeGroup2.wi_inhibitJm.11	:=	NOT GVL1.hxi_alarmInh[43	];
aeGroup2.wi_inhibitJm.12	:=	NOT GVL1.hxi_alarmInh[44	];
aeGroup2.wi_inhibitJm.13	:=	NOT GVL1.hxi_alarmInh[45	];
aeGroup2.wi_inhibitJm.14	:=	NOT GVL1.hxi_alarmInh[46	];
aeGroup2.wi_inhibitJm.15	:=	NOT GVL1.hxi_alarmInh[47	];
			
aeGroup3.wi_inhibitJm.0	:=	NOT GVL1.hxi_alarmInh[48	];
aeGroup3.wi_inhibitJm.1	:=	NOT GVL1.hxi_alarmInh[49	];
aeGroup3.wi_inhibitJm.2	:=	NOT GVL1.hxi_alarmInh[50	];
aeGroup3.wi_inhibitJm.3	:=	NOT GVL1.hxi_alarmInh[51	];
aeGroup3.wi_inhibitJm.4	:=	NOT GVL1.hxi_alarmInh[52	];
aeGroup3.wi_inhibitJm.5	:=	NOT GVL1.hxi_alarmInh[53	];
aeGroup3.wi_inhibitJm.6	:=	NOT GVL1.hxi_alarmInh[54	];
aeGroup3.wi_inhibitJm.7	:=	NOT GVL1.hxi_alarmInh[55	];
aeGroup3.wi_inhibitJm.8	:=	NOT GVL1.hxi_alarmInh[56	];
aeGroup3.wi_inhibitJm.9	:=	NOT GVL1.hxi_alarmInh[57	];
aeGroup3.wi_inhibitJm.10	:=	NOT GVL1.hxi_alarmInh[58	];
aeGroup3.wi_inhibitJm.11	:=	NOT GVL1.hxi_alarmInh[59	];
aeGroup3.wi_inhibitJm.12	:=	NOT GVL1.hxi_alarmInh[60	];
aeGroup3.wi_inhibitJm.13	:=	NOT GVL1.hxi_alarmInh[61	];
aeGroup3.wi_inhibitJm.14	:=	NOT GVL1.hxi_alarmInh[62	];
aeGroup3.wi_inhibitJm.15	:=	NOT GVL1.hxi_alarmInh[63	];
			
aeGroup4.wi_inhibitJm.0	:=	NOT GVL1.hxi_alarmInh[64	];
aeGroup4.wi_inhibitJm.1	:=	NOT GVL1.hxi_alarmInh[65	];
aeGroup4.wi_inhibitJm.2	:=	NOT GVL1.hxi_alarmInh[66	];
aeGroup4.wi_inhibitJm.3	:=	NOT GVL1.hxi_alarmInh[67	];
aeGroup4.wi_inhibitJm.4	:=	NOT GVL1.hxi_alarmInh[68	];
aeGroup4.wi_inhibitJm.5	:=	NOT GVL1.hxi_alarmInh[69	];
aeGroup4.wi_inhibitJm.6	:=	NOT GVL1.hxi_alarmInh[70	];
aeGroup4.wi_inhibitJm.7	:=	NOT GVL1.hxi_alarmInh[71	];
aeGroup4.wi_inhibitJm.8	:=	NOT GVL1.hxi_alarmInh[72	];
aeGroup4.wi_inhibitJm.9	:=	NOT GVL1.hxi_alarmInh[73	];
aeGroup4.wi_inhibitJm.10	:=	NOT GVL1.hxi_alarmInh[74	];
aeGroup4.wi_inhibitJm.11	:=	NOT GVL1.hxi_alarmInh[75	];
aeGroup4.wi_inhibitJm.12	:=	NOT GVL1.hxi_alarmInh[76	];
aeGroup4.wi_inhibitJm.13	:=	NOT GVL1.hxi_alarmInh[77	];
aeGroup4.wi_inhibitJm.14	:=	NOT GVL1.hxi_alarmInh[78	];
aeGroup4.wi_inhibitJm.15	:=	NOT GVL1.hxi_alarmInh[79	];
			
aeGroup5.wi_inhibitJm.0	:=	NOT GVL1.hxi_alarmInh[80	];
aeGroup5.wi_inhibitJm.1	:=	NOT GVL1.hxi_alarmInh[81	];
aeGroup5.wi_inhibitJm.2	:=	NOT GVL1.hxi_alarmInh[82	];
aeGroup5.wi_inhibitJm.3	:=	NOT GVL1.hxi_alarmInh[83	];
aeGroup5.wi_inhibitJm.4	:=	NOT GVL1.hxi_alarmInh[84	];
aeGroup5.wi_inhibitJm.5	:=	NOT GVL1.hxi_alarmInh[85	];
aeGroup5.wi_inhibitJm.6	:=	NOT GVL1.hxi_alarmInh[86	];
aeGroup5.wi_inhibitJm.7	:=	NOT GVL1.hxi_alarmInh[87	];
aeGroup5.wi_inhibitJm.8	:=	NOT GVL1.hxi_alarmInh[88	];
aeGroup5.wi_inhibitJm.9	:=	NOT GVL1.hxi_alarmInh[89	];
aeGroup5.wi_inhibitJm.10	:=	NOT GVL1.hxi_alarmInh[90	];
aeGroup5.wi_inhibitJm.11	:=	NOT GVL1.hxi_alarmInh[91	];
aeGroup5.wi_inhibitJm.12	:=	NOT GVL1.hxi_alarmInh[92	];
aeGroup5.wi_inhibitJm.13	:=	NOT GVL1.hxi_alarmInh[93	];
aeGroup5.wi_inhibitJm.14	:=	NOT GVL1.hxi_alarmInh[94	];
aeGroup5.wi_inhibitJm.15	:=	NOT GVL1.hxi_alarmInh[95	];
			
aeGroup6.wi_inhibitJm.0	:=	NOT GVL1.hxi_alarmInh[96	];
aeGroup6.wi_inhibitJm.1	:=	NOT GVL1.hxi_alarmInh[97	];
aeGroup6.wi_inhibitJm.2	:=	NOT GVL1.hxi_alarmInh[98	];
aeGroup6.wi_inhibitJm.3	:=	NOT GVL1.hxi_alarmInh[99	];
aeGroup6.wi_inhibitJm.4	:=	NOT GVL1.hxi_alarmInh[100	];
aeGroup6.wi_inhibitJm.5	:=	NOT GVL1.hxi_alarmInh[101	];
aeGroup6.wi_inhibitJm.6	:=	NOT GVL1.hxi_alarmInh[102	];
aeGroup6.wi_inhibitJm.7	:=	NOT GVL1.hxi_alarmInh[103	];
aeGroup6.wi_inhibitJm.8	:=	NOT GVL1.hxi_alarmInh[104	];
aeGroup6.wi_inhibitJm.9	:=	NOT GVL1.hxi_alarmInh[105	];
aeGroup6.wi_inhibitJm.10	:=	NOT GVL1.hxi_alarmInh[106	];
aeGroup6.wi_inhibitJm.11	:=	NOT GVL1.hxi_alarmInh[107	];
aeGroup6.wi_inhibitJm.12	:=	NOT GVL1.hxi_alarmInh[108	];
aeGroup6.wi_inhibitJm.13	:=	NOT GVL1.hxi_alarmInh[109	];
aeGroup6.wi_inhibitJm.14	:=	NOT GVL1.hxi_alarmInh[110	];
aeGroup6.wi_inhibitJm.15	:=	NOT GVL1.hxi_alarmInh[111	];
			
aeGroup7.wi_inhibitJm.0	:=	NOT GVL1.hxi_alarmInh[112	];
aeGroup7.wi_inhibitJm.1	:=	NOT GVL1.hxi_alarmInh[113	];
aeGroup7.wi_inhibitJm.2	:=	NOT GVL1.hxi_alarmInh[114	];
aeGroup7.wi_inhibitJm.3	:=	NOT GVL1.hxi_alarmInh[115	];
aeGroup7.wi_inhibitJm.4	:=	NOT GVL1.hxi_alarmInh[116	];
aeGroup7.wi_inhibitJm.5	:=	NOT GVL1.hxi_alarmInh[117	];
aeGroup7.wi_inhibitJm.6	:=	NOT GVL1.hxi_alarmInh[118	];
aeGroup7.wi_inhibitJm.7	:=	NOT GVL1.hxi_alarmInh[119	];
aeGroup7.wi_inhibitJm.8	:=	NOT GVL1.hxi_alarmInh[120	];
aeGroup7.wi_inhibitJm.9	:=	NOT GVL1.hxi_alarmInh[121	];
aeGroup7.wi_inhibitJm.10	:=	NOT GVL1.hxi_alarmInh[122	];
aeGroup7.wi_inhibitJm.11	:=	NOT GVL1.hxi_alarmInh[123	];
aeGroup7.wi_inhibitJm.12	:=	NOT GVL1.hxi_alarmInh[124	];
aeGroup7.wi_inhibitJm.13	:=	NOT GVL1.hxi_alarmInh[125	];
aeGroup7.wi_inhibitJm.14	:=	NOT GVL1.hxi_alarmInh[126	];
aeGroup7.wi_inhibitJm.15	:=	NOT GVL1.hxi_alarmInh[127	];
			
aeGroup8.wi_inhibitJm.0	:=	NOT GVL1.hxi_alarmInh[128	];
aeGroup8.wi_inhibitJm.1	:=	NOT GVL1.hxi_alarmInh[129	];
aeGroup8.wi_inhibitJm.2	:=	NOT GVL1.hxi_alarmInh[130	];
aeGroup8.wi_inhibitJm.3	:=	NOT GVL1.hxi_alarmInh[131	];
aeGroup8.wi_inhibitJm.4	:=	NOT GVL1.hxi_alarmInh[132	];
aeGroup8.wi_inhibitJm.5	:=	NOT GVL1.hxi_alarmInh[133	];
aeGroup8.wi_inhibitJm.6	:=	NOT GVL1.hxi_alarmInh[134	];
aeGroup8.wi_inhibitJm.7	:=	NOT GVL1.hxi_alarmInh[135	];
aeGroup8.wi_inhibitJm.8	:=	NOT GVL1.hxi_alarmInh[136	];
aeGroup8.wi_inhibitJm.9	:=	NOT GVL1.hxi_alarmInh[137	];
aeGroup8.wi_inhibitJm.10	:=	NOT GVL1.hxi_alarmInh[138	];
aeGroup8.wi_inhibitJm.11	:=	NOT GVL1.hxi_alarmInh[139	];
aeGroup8.wi_inhibitJm.12	:=	NOT GVL1.hxi_alarmInh[140	];
aeGroup8.wi_inhibitJm.13	:=	NOT GVL1.hxi_alarmInh[141	];
aeGroup8.wi_inhibitJm.14	:=	NOT GVL1.hxi_alarmInh[142	];
aeGroup8.wi_inhibitJm.15	:=	NOT GVL1.hxi_alarmInh[143	];
			
aeGroup9.wi_inhibitJm.0	:=	NOT GVL1.hxi_alarmInh[144	];
aeGroup9.wi_inhibitJm.1	:=	NOT GVL1.hxi_alarmInh[145	];
aeGroup9.wi_inhibitJm.2	:=	NOT GVL1.hxi_alarmInh[146	];
aeGroup9.wi_inhibitJm.3	:=	NOT GVL1.hxi_alarmInh[147	];
aeGroup9.wi_inhibitJm.4	:=	NOT GVL1.hxi_alarmInh[148	];
aeGroup9.wi_inhibitJm.5	:=	NOT GVL1.hxi_alarmInh[149	];
aeGroup9.wi_inhibitJm.6	:=	NOT GVL1.hxi_alarmInh[150	];
aeGroup9.wi_inhibitJm.7	:=	NOT GVL1.hxi_alarmInh[151	];
aeGroup9.wi_inhibitJm.8	:=	NOT GVL1.hxi_alarmInh[152	];
aeGroup9.wi_inhibitJm.9	:=	NOT GVL1.hxi_alarmInh[153	];
aeGroup9.wi_inhibitJm.10	:=	NOT GVL1.hxi_alarmInh[154	];
aeGroup9.wi_inhibitJm.11	:=	NOT GVL1.hxi_alarmInh[155	];
aeGroup9.wi_inhibitJm.12	:=	NOT GVL1.hxi_alarmInh[156	];
aeGroup9.wi_inhibitJm.13	:=	NOT GVL1.hxi_alarmInh[157	];
aeGroup9.wi_inhibitJm.14	:=	NOT GVL1.hxi_alarmInh[158	];
aeGroup9.wi_inhibitJm.15	:=	NOT GVL1.hxi_alarmInh[159	];
			
aeGroup10.wi_inhibitJm.0	:=	NOT GVL1.hxi_alarmInh[160	];
aeGroup10.wi_inhibitJm.1	:=	NOT GVL1.hxi_alarmInh[161	];
aeGroup10.wi_inhibitJm.2	:=	NOT GVL1.hxi_alarmInh[162	];
aeGroup10.wi_inhibitJm.3	:=	NOT GVL1.hxi_alarmInh[163	];
aeGroup10.wi_inhibitJm.4	:=	NOT GVL1.hxi_alarmInh[164	];
aeGroup10.wi_inhibitJm.5	:=	NOT GVL1.hxi_alarmInh[165	];
aeGroup10.wi_inhibitJm.6	:=	NOT GVL1.hxi_alarmInh[166	];
aeGroup10.wi_inhibitJm.7	:=	NOT GVL1.hxi_alarmInh[167	];
aeGroup10.wi_inhibitJm.8	:=	NOT GVL1.hxi_alarmInh[168	];
aeGroup10.wi_inhibitJm.9	:=	NOT GVL1.hxi_alarmInh[169	];
aeGroup10.wi_inhibitJm.10	:=	NOT GVL1.hxi_alarmInh[170	];
aeGroup10.wi_inhibitJm.11	:=	NOT GVL1.hxi_alarmInh[171	];
aeGroup10.wi_inhibitJm.12	:=	NOT GVL1.hxi_alarmInh[172	];
aeGroup10.wi_inhibitJm.13	:=	NOT GVL1.hxi_alarmInh[173	];
aeGroup10.wi_inhibitJm.14	:=	NOT GVL1.hxi_alarmInh[174	];
aeGroup10.wi_inhibitJm.15	:=	NOT GVL1.hxi_alarmInh[175	];
			
aeGroup11.wi_inhibitJm.0	:=	NOT GVL1.hxi_alarmInh[176	];
aeGroup11.wi_inhibitJm.1	:=	NOT GVL1.hxi_alarmInh[177	];
aeGroup11.wi_inhibitJm.2	:=	NOT GVL1.hxi_alarmInh[178	];
aeGroup11.wi_inhibitJm.3	:=	NOT GVL1.hxi_alarmInh[179	];
aeGroup11.wi_inhibitJm.4	:=	NOT GVL1.hxi_alarmInh[180	];
aeGroup11.wi_inhibitJm.5	:=	NOT GVL1.hxi_alarmInh[181	];
aeGroup11.wi_inhibitJm.6	:=	NOT GVL1.hxi_alarmInh[182	];
aeGroup11.wi_inhibitJm.7	:=	NOT GVL1.hxi_alarmInh[183	];
aeGroup11.wi_inhibitJm.8	:=	NOT GVL1.hxi_alarmInh[184	];
aeGroup11.wi_inhibitJm.9	:=	NOT GVL1.hxi_alarmInh[185	];
aeGroup11.wi_inhibitJm.10	:=	NOT GVL1.hxi_alarmInh[186	];
aeGroup11.wi_inhibitJm.11	:=	NOT GVL1.hxi_alarmInh[187	];
aeGroup11.wi_inhibitJm.12	:=	NOT GVL1.hxi_alarmInh[188	];
aeGroup11.wi_inhibitJm.13	:=	NOT GVL1.hxi_alarmInh[189	];
aeGroup11.wi_inhibitJm.14	:=	NOT GVL1.hxi_alarmInh[190	];
aeGroup11.wi_inhibitJm.15	:=	NOT GVL1.hxi_alarmInh[191	];
			
aeGroup12.wi_inhibitJm.0	:=	NOT GVL1.hxi_alarmInh[192	];
aeGroup12.wi_inhibitJm.1	:=	NOT GVL1.hxi_alarmInh[193	];
aeGroup12.wi_inhibitJm.2	:=	NOT GVL1.hxi_alarmInh[194	];
aeGroup12.wi_inhibitJm.3	:=	NOT GVL1.hxi_alarmInh[195	];
aeGroup12.wi_inhibitJm.4	:=	NOT GVL1.hxi_alarmInh[196	];
aeGroup12.wi_inhibitJm.5	:=	NOT GVL1.hxi_alarmInh[197	];
aeGroup12.wi_inhibitJm.6	:=	NOT GVL1.hxi_alarmInh[198	];
aeGroup12.wi_inhibitJm.7	:=	NOT GVL1.hxi_alarmInh[199	];
aeGroup12.wi_inhibitJm.8	:=	NOT GVL1.hxi_alarmInh[200	];
aeGroup12.wi_inhibitJm.9	:=	NOT GVL1.hxi_alarmInh[201	];
aeGroup12.wi_inhibitJm.10	:=	NOT GVL1.hxi_alarmInh[202	];
aeGroup12.wi_inhibitJm.11	:=	NOT GVL1.hxi_alarmInh[203	];
aeGroup12.wi_inhibitJm.12	:=	NOT GVL1.hxi_alarmInh[204	];
aeGroup12.wi_inhibitJm.13	:=	NOT GVL1.hxi_alarmInh[205	];
aeGroup12.wi_inhibitJm.14	:=	NOT GVL1.hxi_alarmInh[206	];
aeGroup12.wi_inhibitJm.15	:=	NOT GVL1.hxi_alarmInh[207	];
			
tmGroup0.wi_chParaJm.0	:=	NOT GVL1.hxi_alarmInh[208	];
tmGroup0.wi_chParaJm.1	:=	NOT GVL1.hxi_alarmInh[209	];
tmGroup0.wi_chParaJm.2	:=	NOT GVL1.hxi_alarmInh[210	];
tmGroup0.wi_chParaJm.3	:=	NOT GVL1.hxi_alarmInh[211	];
tmGroup0.wi_chParaJm.4	:=	NOT GVL1.hxi_alarmInh[212	];
tmGroup0.wi_chParaJm.10	:=	NOT GVL1.hxi_alarmInh[213	];
			
tmGroup1.wi_chParaJm.0	:=	NOT GVL1.hxi_alarmInh[214	];
tmGroup1.wi_chParaJm.1	:=	NOT GVL1.hxi_alarmInh[215	];
tmGroup1.wi_chParaJm.2	:=	NOT GVL1.hxi_alarmInh[216	];
tmGroup1.wi_chParaJm.3	:=	NOT GVL1.hxi_alarmInh[217	];
tmGroup1.wi_chParaJm.4	:=	NOT GVL1.hxi_alarmInh[218	];
tmGroup1.wi_chParaJm.10	:=	NOT GVL1.hxi_alarmInh[219	];
			
tmGroup2.wi_chParaJm.0	:=	NOT GVL1.hxi_alarmInh[220	];
tmGroup2.wi_chParaJm.1	:=	NOT GVL1.hxi_alarmInh[221	];
tmGroup2.wi_chParaJm.2	:=	NOT GVL1.hxi_alarmInh[222	];
tmGroup2.wi_chParaJm.3	:=	NOT GVL1.hxi_alarmInh[223	];
tmGroup2.wi_chParaJm.4	:=	NOT GVL1.hxi_alarmInh[224	];
tmGroup2.wi_chParaJm.10	:=	NOT GVL1.hxi_alarmInh[225	];
			
tmGroup3.wi_chParaJm.0	:=	NOT GVL1.hxi_alarmInh[226	];
tmGroup3.wi_chParaJm.1	:=	NOT GVL1.hxi_alarmInh[227	];
tmGroup3.wi_chParaJm.2	:=	NOT GVL1.hxi_alarmInh[228	];
tmGroup3.wi_chParaJm.3	:=	NOT GVL1.hxi_alarmInh[229	];
tmGroup3.wi_chParaJm.4	:=	NOT GVL1.hxi_alarmInh[230	];
tmGroup3.wi_chParaJm.10	:=	NOT GVL1.hxi_alarmInh[231	];
			
tmGroup4.wi_chParaJm.0	:=	NOT GVL1.hxi_alarmInh[232	];
tmGroup4.wi_chParaJm.1	:=	NOT GVL1.hxi_alarmInh[233	];
tmGroup4.wi_chParaJm.2	:=	NOT GVL1.hxi_alarmInh[234	];
tmGroup4.wi_chParaJm.3	:=	NOT GVL1.hxi_alarmInh[235	];
tmGroup4.wi_chParaJm.4	:=	NOT GVL1.hxi_alarmInh[236	];
tmGroup4.wi_chParaJm.10	:=	NOT GVL1.hxi_alarmInh[237	];
			
tmGroup5.wi_chParaJm.0	:=	NOT GVL1.hxi_alarmInh[238	];
tmGroup5.wi_chParaJm.1	:=	NOT GVL1.hxi_alarmInh[239	];
tmGroup5.wi_chParaJm.2	:=	NOT GVL1.hxi_alarmInh[240	];
tmGroup5.wi_chParaJm.3	:=	NOT GVL1.hxi_alarmInh[241	];
tmGroup5.wi_chParaJm.4	:=	NOT GVL1.hxi_alarmInh[242	];
tmGroup5.wi_chParaJm.10	:=	NOT GVL1.hxi_alarmInh[243	];
			
tmGroup6.wi_chParaJm.0	:=	NOT GVL1.hxi_alarmInh[244	];
tmGroup6.wi_chParaJm.1	:=	NOT GVL1.hxi_alarmInh[245	];
tmGroup6.wi_chParaJm.2	:=	NOT GVL1.hxi_alarmInh[246	];
tmGroup6.wi_chParaJm.3	:=	NOT GVL1.hxi_alarmInh[247	];
tmGroup6.wi_chParaJm.4	:=	NOT GVL1.hxi_alarmInh[248	];
tmGroup6.wi_chParaJm.10	:=	NOT GVL1.hxi_alarmInh[249	];
			
tmGroup7.wi_chParaJm.0	:=	NOT GVL1.hxi_alarmInh[250	];
tmGroup7.wi_chParaJm.1	:=	NOT GVL1.hxi_alarmInh[251	];
tmGroup7.wi_chParaJm.2	:=	NOT GVL1.hxi_alarmInh[252	];
tmGroup7.wi_chParaJm.3	:=	NOT GVL1.hxi_alarmInh[253	];
tmGroup7.wi_chParaJm.4	:=	NOT GVL1.hxi_alarmInh[254	];
tmGroup7.wi_chParaJm.10	:=	NOT GVL1.hxi_alarmInh[255	];
			
tmGroup8.wi_chParaJm.0	:=	NOT GVL1.hxi_alarmInh[256	];
tmGroup8.wi_chParaJm.1	:=	NOT GVL1.hxi_alarmInh[257	];
tmGroup8.wi_chParaJm.2	:=	NOT GVL1.hxi_alarmInh[258	];
tmGroup8.wi_chParaJm.3	:=	NOT GVL1.hxi_alarmInh[259	];
tmGroup8.wi_chParaJm.4	:=	NOT GVL1.hxi_alarmInh[260	];
tmGroup8.wi_chParaJm.10	:=	NOT GVL1.hxi_alarmInh[261	];
			
tmGroup9.wi_chParaJm.0	:=	NOT GVL1.hxi_alarmInh[262	];
tmGroup9.wi_chParaJm.1	:=	NOT GVL1.hxi_alarmInh[263	];
tmGroup9.wi_chParaJm.2	:=	NOT GVL1.hxi_alarmInh[264	];
tmGroup9.wi_chParaJm.3	:=	NOT GVL1.hxi_alarmInh[265	];
tmGroup9.wi_chParaJm.4	:=	NOT GVL1.hxi_alarmInh[266	];
tmGroup9.wi_chParaJm.10	:=	NOT GVL1.hxi_alarmInh[267	];
			
tmGroup10.wi_chParaJm.0	:=	NOT GVL1.hxi_alarmInh[268	];
tmGroup10.wi_chParaJm.1	:=	NOT GVL1.hxi_alarmInh[269	];
tmGroup10.wi_chParaJm.2	:=	NOT GVL1.hxi_alarmInh[270	];
tmGroup10.wi_chParaJm.3	:=	NOT GVL1.hxi_alarmInh[271	];
tmGroup10.wi_chParaJm.4	:=	NOT GVL1.hxi_alarmInh[272	];
tmGroup10.wi_chParaJm.10	:=	NOT GVL1.hxi_alarmInh[273	];
			
tmGroup11.wi_chParaJm.0	:=	NOT GVL1.hxi_alarmInh[274	];
tmGroup11.wi_chParaJm.1	:=	NOT GVL1.hxi_alarmInh[275	];
tmGroup11.wi_chParaJm.2	:=	NOT GVL1.hxi_alarmInh[276	];
tmGroup11.wi_chParaJm.3	:=	NOT GVL1.hxi_alarmInh[277	];
tmGroup11.wi_chParaJm.4	:=	NOT GVL1.hxi_alarmInh[278	];
tmGroup11.wi_chParaJm.10	:=	NOT GVL1.hxi_alarmInh[279	];
			
tmGroup12.wi_chParaJm.0	:=	NOT GVL1.hxi_alarmInh[280	];
tmGroup12.wi_chParaJm.1	:=	NOT GVL1.hxi_alarmInh[281	];
tmGroup12.wi_chParaJm.2	:=	NOT GVL1.hxi_alarmInh[282	];
tmGroup12.wi_chParaJm.3	:=	NOT GVL1.hxi_alarmInh[283	];
tmGroup12.wi_chParaJm.4	:=	NOT GVL1.hxi_alarmInh[284	];
tmGroup12.wi_chParaJm.10	:=	NOT GVL1.hxi_alarmInh[285	];
			
tmGroup13.wi_chParaJm.0	:=	NOT GVL1.hxi_alarmInh[286	];
tmGroup13.wi_chParaJm.1	:=	NOT GVL1.hxi_alarmInh[287	];
tmGroup13.wi_chParaJm.2	:=	NOT GVL1.hxi_alarmInh[288	];
tmGroup13.wi_chParaJm.3	:=	NOT GVL1.hxi_alarmInh[289	];
tmGroup13.wi_chParaJm.4	:=	NOT GVL1.hxi_alarmInh[290	];
tmGroup13.wi_chParaJm.10	:=	NOT GVL1.hxi_alarmInh[291	];
			
tmGroup14.wi_chParaJm.0	:=	NOT GVL1.hxi_alarmInh[292	];
tmGroup14.wi_chParaJm.1	:=	NOT GVL1.hxi_alarmInh[293	];
tmGroup14.wi_chParaJm.2	:=	NOT GVL1.hxi_alarmInh[294	];
tmGroup14.wi_chParaJm.3	:=	NOT GVL1.hxi_alarmInh[295	];
tmGroup14.wi_chParaJm.4	:=	NOT GVL1.hxi_alarmInh[296	];
tmGroup14.wi_chParaJm.5	:=	NOT GVL1.hxi_alarmInh[297	];
			
tmGroup15.wi_chParaJm.0	:=	NOT GVL1.hxi_alarmInh[298	];
tmGroup15.wi_chParaJm.1	:=	NOT GVL1.hxi_alarmInh[299	];
tmGroup15.wi_chParaJm.2	:=	NOT GVL1.hxi_alarmInh[300	];
tmGroup15.wi_chParaJm.3	:=	NOT GVL1.hxi_alarmInh[301	];
tmGroup15.wi_chParaJm.4	:=	NOT GVL1.hxi_alarmInh[302	];
tmGroup15.wi_chParaJm.5	:=	NOT GVL1.hxi_alarmInh[303	];
END_ACTION

ACTION smart_ship:
JB1_DATA.0	 := GVL1.hwo_digitalAlarms[0].0	;	(*	DI:01	GEN.ROOM PORT BILGE ALARM	*)
JB1_DATA.1	 := GVL1.hwo_digitalAlarms[0].1	;	(*	DI:02	PORT GEN EXHAUST TEMP HIGH	*)
JB1_DATA.2	 := GVL1.hwo_digitalAlarms[0].2	;	(*	DI:03	PORT GENERATOR COMMON ALARM	*)
JB1_DATA.3	 := GVL1.hwo_digitalEvents[0].3	;	(*	DI:04	PORT GENERATOR RUNNING INDICATION	*)
JB1_DATA.4	 := GVL1.hwo_digitalAlarms[0].4	;	(*	DI:05	A.FOULING ALARM: DG(P) & EMG FIRE.P S/C 	*)
JB1_DATA.5	 := GVL1.hwo_digitalAlarms[0].5	;	(*	DI:06	STEERING CP: PHASE FAIL MOTOR 1	*)
JB1_DATA.6	 := GVL1.hwo_digitalAlarms[0].6	;	(*	DI:07	STEERING CP: POWER FAIL MOTOR 1	*)
JB1_DATA.7	 := GVL1.hwo_digitalAlarms[0].7	;	(*	DI:08	STEERING CP: CONTROL FAIL MOTOR 1	*)
JB1_DATA.8	 := GVL1.hwo_digitalAlarms[0].8	;	(*	DI:09	STEERING CP: OVERLOAD MOTOR 1	*)
JB1_DATA.9	 := GVL1.hwo_digitalAlarms[0].9	;	(*	DI:10	STEERING CP: PHASE FAIL MOTOR 2	*)
JB1_DATA.10	 := GVL1.hwo_digitalAlarms[0].10	;	(*	DI:11	STEERING CP: POWER FAIL MOTOR 2	*)
JB1_DATA.11	 := GVL1.hwo_digitalAlarms[0].11	;	(*	DI:12	STEERING CP: CONTROL FAIL MOTOR 2	*)
JB1_DATA.12	 := GVL1.hwo_digitalAlarms[0].12	;	(*	DI:13	STEERING CP: OVERLOAD MOTOR 2	*)
JB1_DATA.13	 := GVL1.hwo_digitalAlarms[0].13	;	(*	DI:14	STEERING CP: LOW OIL LEVEL ALARM	*)
JB1_DATA.14	 := GVL1.hwo_digitalAlarms[0].14	;	(*	DI:15	STEERING CP: HIGH OIL TEMP ALARM	*)
JB1_DATA.15	 := GVL1.hwo_digitalAlarms[0].15	;	(*	DI:16	STEERING CP: LOW OIL PRESSURE ALARM	*)
						
JB2_DATA.0	 := GVL1.hwo_digitalAlarms[1].0	;	(*	DI:17	GEN.ROOM STBD BILGE ALARM	*)
JB2_DATA.1	 := GVL1.hwo_digitalEvents[1].1	;	(*	DI:18	ENGINE ROOM AFT WT DOOR	*)
JB2_DATA.2	 := GVL1.hwo_digitalAlarms[1].2	;	(*	DI:19	CENTER ME EXHAUST TEMP HIGH	*)
JB2_DATA.3	 := GVL1.hwo_digitalAlarms[1].3	;	(*	DI:20	STBD GEN EXHAUST TEMP HIGH	*)
JB2_DATA.4	 := GVL1.hwo_digitalAlarms[1].4	;	(*	DI:21	STBD GENERATOR COMMON ALARM	*)
JB2_DATA.5	 := GVL1.hwo_digitalEvents[1].5	;	(*	DI:22	STBD GENERATOR RUNNING INDICATION	*)
JB2_DATA.6	 := GVL1.hwo_digitalAlarms[1].6	;	(*	DI:23	STBD ME EXHAUST TEMP HIGH	*)
JB2_DATA.7	 := GVL1.hwo_digitalAlarms[1].7	;	(*	DI:24	BOW THRUSTER COMMON ALARM	*)
JB2_DATA.8	 := GVL1.hwo_digitalAlarms[1].8	;	(*	DI:25	BOW THRUSTER LOW OIL LEVEL ALARM	*)
JB2_DATA.9	 := GVL1.hwo_digitalAlarms[1].9	;	(*	DI:26	BOW THRUSTER HIGH OIL TEMP ALARM	*)
JB2_DATA.10	 := GVL1.hwo_digitalAlarms[1].10	;	(*	DI:27	OWS POWER SUPPLY FAILURE	*)
JB2_DATA.11	 := GVL1.hwo_digitalAlarms[1].11	;	(*	DI:28	OWS 15 PPM ALARM	*)
JB2_DATA.12	 := GVL1.hwo_digitalAlarms[1].12	;	(*	DI:29	DCDB-2 BATTERY BREAKER TRIP ALARM	*)
JB2_DATA.13	 := GVL1.hwo_digitalAlarms[1].13	;	(*	DI:30	DCDB-2 EARTH FAULT ALARM	*)
JB2_DATA.14	 := GVL1.hwo_digitalAlarms[1].14	;	(*	DI:31	DCDB-2 BATTERY CHARGER FAIL ALARM	*)
JB2_DATA.15	 := GVL1.hwo_digitalAlarms[1].15	;	(*	DI:32	DCDB-2 BATTERY DISCHARGE ALARM	*)
						
JB3_DATA.0	 := GVL1.hwo_digitalAlarms[2].0	;	(*	DI:33	PORT STERN TUBE FLOW ALARM	*)
JB3_DATA.1	 := GVL1.hwo_digitalAlarms[2].1	;	(*	DI:34	STBD STERN TUBE FLOW ALARM	*)
JB3_DATA.2	 := GVL1.hwo_digitalAlarms[2].2	;	(*	DI:35	CENTER STERN TUBE FLOW ALARM	*)
JB3_DATA.3	 := GVL1.hwo_digitalAlarms[2].3	;	(*	DI:36	PORT ME EXHAUST TEMP HIGH	*)
JB3_DATA.4	 := GVL1.hwo_digitalAlarms[2].4	;	(*	DI:37	A.FOULING ALARM: AUX SW.P &  FIRE.P S/C	*)
JB3_DATA.5	 := GVL1.hwo_digitalAlarms[2].5	;	(*	DI:38	A.FOULING ALARM: DG(S) S/C	*)
JB3_DATA.6	 := GVL1.hwo_digitalAlarms[2].6	;	(*	DI:39	PORT ME/GEN STARTING BATTERY LOW ALARM	*)
JB3_DATA.7	 := GVL1.hwo_digitalAlarms[2].7	;	(*	DI:40	STBD ME/GEN STARTING BATTERY LOW ALARM	*)
JB3_DATA.8	 := GVL1.hwo_digitalAlarms[2].8	;	(*	DI:41	CENTER ME STARTING BATTERY LOW ALARM	*)
JB3_DATA.9	 := GVL1.hwo_digitalEvents[2].9	;	(*	DI:42	AUX COOLING PUMP-2 RUNNING	*)
JB3_DATA.10	 := GVL1.hwo_digitalAlarms[2].10	;	(*	DI:43	AUX COOLING PUMP-2 TRIP	*)
JB3_DATA.11	 := GVL1.hwo_digitalAlarms[2].11	;	(*	DI:44	ENG.ROOM AFT BILGE ALARM	*)
JB3_DATA.12	 := GVL1.hwo_digitalAlarms[2].12	;	(*	DI:45	ENG.ROOM AFT FLOOD ALARM	*)
JB3_DATA.13	 := GVL1.hwo_digitalAlarms[2].13	;	(*	DI:46	SPARE	*)
JB3_DATA.14	 := GVL1.hwo_digitalAlarms[2].14	;	(*	DI:47	SPARE	*)
JB3_DATA.15	 := GVL1.hwo_digitalAlarms[2].15	;	(*	DI:48	SPARE	*)
						
JB4_DATA.0	 := GVL1.hwo_digitalAlarms[3].0	;	(*	DI:49	ENG.ROOM FWD BILGE ALARM	*)
JB4_DATA.1	 := GVL1.hwo_digitalAlarms[3].1	;	(*	DI:50	ENG.ROOM FWD FLOOD ALARM	*)
JB4_DATA.2	 := GVL1.hwo_digitalEvents[3].2	;	(*	DI:51	ENGINE ROOM FWD WT DOOR	*)
JB4_DATA.3	 := GVL1.hwo_digitalAlarms[3].3	;	(*	DI:52	PROPULSION SYSTEM POWER SUPPLY FAIL	*)
JB4_DATA.4	 := GVL1.hwo_digitalAlarms[3].4	;	(*	DI:53	PORT ME PROP.MODULE COMMON ALARM	*)
JB4_DATA.5	 := GVL1.hwo_digitalAlarms[3].5	;	(*	DI:54	STBD ME PROP.MODULE COMMON ALARM	*)
JB4_DATA.6	 := GVL1.hwo_digitalAlarms[3].6	;	(*	DI:55	CENTER ME PROP.MODULE COMMON ALARM	*)
JB4_DATA.7	 := GVL1.hwo_digitalAlarms[3].7	;	(*	DI:56	A.FOULING ALARM: PORT ME & STBD ME S/C	*)
JB4_DATA.8	 := GVL1.hwo_digitalAlarms[3].8	;	(*	DI:57	A.FOULING ALARM: CENETR ME S/C	*)
JB4_DATA.9	 := GVL1.hwo_digitalAlarms[3].9	;	(*	DI:58	A.FOULING ALARM: SW DOMESTIC & A/C.P SC	*)
JB4_DATA.10	 := GVL1.hwo_digitalAlarms[3].10	;	(*	DI:59	ENG.ROOM CO2 RELEASE EAVC ALARM	*)
JB4_DATA.11	 := GVL1.hwo_digitalAlarms[3].11	;	(*	DI:60	GEN.ROOM CO2 RELEASE EVAC ALARM	*)
JB4_DATA.12	 := GVL1.hwo_digitalAlarms[3].12	;	(*	DI:61	CO2 LEAKAGE ALARM	*)
JB4_DATA.13	 := GVL1.hwo_digitalAlarms[3].13	;	(*	DI:62	ENG ROOM CO2 RELEASED ALARM	*)
JB4_DATA.14	 := GVL1.hwo_digitalAlarms[3].14	;	(*	DI:63	GEN ROOM CO2 RELEASED ALARM	*)
JB4_DATA.15	 := GVL1.hwo_digitalAlarms[3].15	;	(*	DI:64	CO2 SYSTEM POWER FAIL ALARM	*)
						
JB5_DATA.0	 := GVL1.hwo_digitalAlarms[4].0	;	(*	DI:65	PUMP ROOM AFT PORT BILGE ALARM	*)
JB5_DATA.1	 := GVL1.hwo_digitalAlarms[4].1	;	(*	DI:66	PUMP ROOM AFT STBD BILGE ALARM	*)
JB5_DATA.2	 := GVL1.hwo_digitalAlarms[4].2	;	(*	DI:67	V.SPACE PUMP ROOM FWD (P) BILGE ALARM	*)
JB5_DATA.3	 := GVL1.hwo_digitalAlarms[4].3	;	(*	DI:68	V.SPACE PUMP ROOM FWD (S) BILGE ALARM	*)
JB5_DATA.4	 := GVL1.hwo_digitalAlarms[4].4	;	(*	DI:69	ACCOM.AREA AFT BILGE ALARM	*)
JB5_DATA.5	 := GVL1.hwo_digitalEvents[4].5	;	(*	DI:70	PUMP ROOM FWD WT DOOR	*)
JB5_DATA.6	 := GVL1.hwo_digitalAlarms[4].6	;	(*	DI:71	STP OVERFLOW ALARM	*)
JB5_DATA.7	 := GVL1.hwo_digitalAlarms[4].7	;	(*	DI:72	A/C SYSTEM COMMON ALARM	*)
JB5_DATA.8	 := GVL1.hwo_digitalAlarms[4].8	;	(*	DI:73	ACCOM.AREA FWD BILGE ALARM	*)
JB5_DATA.9	 := GVL1.hwo_digitalAlarms[4].9	;	(*	DI:74	FWD PASSAGE BILGE ALARM	*)
JB5_DATA.10	 := GVL1.hwo_digitalAlarms[4].10	;	(*	DI:75	FOREPEAK COMPT BILGE ALARM	*)
JB5_DATA.11	 := GVL1.hwo_digitalEvents[4].11	;	(*	DI:76	ACCOM.AREA WT DOOR	*)
JB5_DATA.12	 := GVL1.hwo_digitalAlarms[4].12	;	(*	DI:77	A/C FIRE DAMPER CLOSED ALARM	*)
JB5_DATA.13	 := GVL1.hwo_digitalAlarms[4].13	;	(*	DI:78	GALLEY VENT OUT FIRE DAMPER CLOSED ALARM	*)
JB5_DATA.14	 := GVL1.hwo_digitalAlarms[4].14	;	(*	DI:79	GALLEY VENT IN FIRE DAMPER CLOSED ALARM	*)
JB5_DATA.15	 := GVL1.hwo_digitalAlarms[4].15	;	(*	DI:80	GALLEY HD VENT FIRE DAMPER CLOSED ALARM	*)
						
JB6_DATA.0	 := GVL1.hwo_digitalAlarms[5].0	;	(*	DI:81	DCDB1 SEC-1 BAT.CHARGER FAILURE ALARM	*)
JB6_DATA.1	 := GVL1.hwo_digitalAlarms[5].1	;	(*	DI:82	DCDB1 SEC-1 BAT. DISCHARGE ALARM	*)
JB6_DATA.2	 := GVL1.hwo_digitalAlarms[5].2	;	(*	DI:83	DCDB1 SEC-1 BAT. LOW VOLT ALARM	*)
JB6_DATA.3	 := GVL1.hwo_digitalAlarms[5].3	;	(*	DI:84	DCDB1 SEC-1 BAT. BANK CB TRIP ALARM	*)
JB6_DATA.4	 := GVL1.hwo_digitalAlarms[5].4	;	(*	DI:85	DCDB1 SEC-2 BAT.CHARGER FAILURE ALARM	*)
JB6_DATA.5	 := GVL1.hwo_digitalAlarms[5].5	;	(*	DI:86	DCDB1 SEC-2 BAT. DISCHARGE ALARM	*)
JB6_DATA.6	 := GVL1.hwo_digitalAlarms[5].6	;	(*	DI:87	DCDB1 SEC-2 BAT. LOW VOLT ALARM	*)
JB6_DATA.7	 := GVL1.hwo_digitalAlarms[5].7	;	(*	DI:88	DCDB1 SEC-2 BAT. BANK CB TRIP ALARM	*)
JB6_DATA.8	 := GVL1.hwo_digitalAlarms[5].8	;	(*	DI:89	SEC-1 AND SEC-2 EARTH FAULT	*)
JB6_DATA.9	 := GVL1.hwo_digitalAlarms[5].9	;	(*	DI:90	FREEZER CTRL PANEL COMMON ALARM	*)
JB6_DATA.10	 := GVL1.hwo_digitalAlarms[5].10	;	(*	DI:91	CHILLER CTRL PANEL COMMON ALARM	*)
JB6_DATA.11	 := GVL1.hwo_digitalAlarms[5].11	;	(*	DI:92	MAN TRAP ALARM: FREEZER ROOM	*)
JB6_DATA.12	 := GVL1.hwo_digitalAlarms[5].12	;	(*	DI:93	MAN TRAP ALARM: CHILLER ROOM	*)
JB6_DATA.13	 := GVL1.hwo_digitalAlarms[5].13	;	(*	DI:94	PUMP RM COMP. AREA AREA REF. LEAKAGE ALARM 	*)
JB6_DATA.14	 := GVL1.hwo_digitalAlarms[5].14	;	(*	DI:95	BELOW DECK. AREA AREA REF. LEAKAGE ALARM 	*)
JB6_DATA.15	 := GVL1.hwo_digitalAlarms[5].15	;	(*	DI:96	CO2 ROOM FAN TRIP ALARM	*)
						
